// TIA Portal V20 export
FUNCTION_BLOCK "CallEquipment"   // FB44, LAD
TITLE = CallEquipment
AUTHOR : ERsystem_FA2_DH. Kim
// This block contains the logic and futher calls (e.g. sequences, control modules, diagnostics etc.) of the equipment module.
// stored: IsIECCheckEnabled true, MemoryReserve 100, Namespace Unit1.Em7, SetENOAutomatically false
   VAR_INPUT
      ZoneOperationEnable { ExternalWritable := 'False'} : "LWONIK_typeSafetyZoneManualOperation";
   END_VAR
   VAR_IN_OUT
      unitStatus : "LAF_typeUnitStatus";   // Current unit status o be used in this EM
      emFeedback : "LUC_typeEmFeedback";   // Feedback of the EM to the Unit
      unitAlarmDB : "LAF_typeAlarms";   // Summarized EM Alarms for the Unit
   END_VAR
   VAR
      instSequenceSepaClamp { ExternalAccessible := 'False'; ExternalVisible := 'False'; ExternalWritable := 'False'} : "Unit1.Em7.Sequence_1_SepaClamp";
      instSequenceSepaGripper { ExternalAccessible := 'False'; ExternalVisible := 'False'; ExternalWritable := 'False'} : "Unit1.Em7.Sequence_2_SepaGripper";
      instSequenceJellyRollWinder { ExternalAccessible := 'False'; ExternalVisible := 'False'; ExternalWritable := 'False'} : "Unit1.Em7.Sequence_3_JellyRollWinder";
      instSepaClampHomeJob1 { S7_SetPoint := 'True'} : "LAF_SelectJob";
      instSepaClampLoadJob2 { S7_SetPoint := 'True'} : "LAF_SelectJob";
      instSepaClampUnloadJob3 { S7_SetPoint := 'True'} : "LAF_SelectJob";
      instSepaClampUnloadCamJob10 { S7_SetPoint := 'True'} : "LAF_SelectJob";
      instSepaClampUnloadStopSyncJob11 { S7_SetPoint := 'True'} : "LAF_SelectJob";
      instSepaClampUnloadReturnJob12 { S7_SetPoint := 'True'} : "LAF_SelectJob";
      instSepaGripperHomeJob1 { S7_SetPoint := 'True'} : "LAF_SelectJob";
      instSepaGripperGripReadyJob2 { S7_SetPoint := 'True'} : "LAF_SelectJob";
      instSepaGripperGripSepaTailJob3 { S7_SetPoint := 'True'} : "LAF_SelectJob";
      instSepaGripperWinderMoveJob4 { S7_SetPoint := 'True'} : "LAF_SelectJob";
      instSepaGripperJellyRollUnGripJob5 { S7_SetPoint := 'True'} : "LAF_SelectJob";
      instSepaGripperJellyRollGripJob6 { S7_SetPoint := 'True'} : "LAF_SelectJob";
      instSepaGripperUnloadReadyJob7 { S7_SetPoint := 'True'} : "LAF_SelectJob";
      instSepaGripperUnloadJob8 { S7_SetPoint := 'True'} : "LAF_SelectJob";
      instSepaGripperReturnJob9 { S7_SetPoint := 'True'} : "LAF_SelectJob";
      instSepaGripperGripReadyJob11 { S7_SetPoint := 'True'} : "LAF_SelectJob";
      instSepaGripperLoadToStackTableJob12 { S7_SetPoint := 'True'} : "LAF_SelectJob";
      instSepaGripperUnLoadToJellyRollWinderJob14 { S7_SetPoint := 'True'} : "LAF_SelectJob";
      instSepaGripperLoadToJellyRollWinderJob15 { S7_SetPoint := 'True'} : "LAF_SelectJob";
      instSepaGripperUnloadToInspectionJob17 { S7_SetPoint := 'True'} : "LAF_SelectJob";
      instSepaGripperReturnJob18 { S7_SetPoint := 'True'} : "LAF_SelectJob";
      instJellyRollWinderHomeJob1 { S7_SetPoint := 'True'} : "LAF_SelectJob";
      instJellyRollWinderLoadJob2 { S7_SetPoint := 'True'} : "LAF_SelectJob";
      instJellyRollWinderWinding1Job3 { S7_SetPoint := 'True'} : "LAF_SelectJob";
      instJellyRollWinderPusherReadyJob4 { S7_SetPoint := 'True'} : "LAF_SelectJob";
      instJellyRollWinderWinding2Job5 { S7_SetPoint := 'True'} : "LAF_SelectJob";
      instJellyRollWinderUnloadJob6 { S7_SetPoint := 'True'} : "LAF_SelectJob";
      instJellyRollWinderCamWinding1stJob10 { S7_SetPoint := 'True'} : "LAF_SelectJob";
      instJellyRollWinderCamPusherReadyJob11 { S7_SetPoint := 'True'} : "LAF_SelectJob";
      instJellyRollWinderCamStartSyncJob12 { S7_SetPoint := 'True'} : "LAF_SelectJob";
      instJellyRollWinderCamWinding2ndJob13 { S7_SetPoint := 'True'} : "LAF_SelectJob";
      instJellyRollWinderCamStopSyncJob14 { S7_SetPoint := 'True'} : "LAF_SelectJob";
      instCmSepaClampDetectSensor { ExternalAccessible := 'False'; ExternalVisible := 'False'; ExternalWritable := 'False'} : "LBC_DigitalSignalCn";
      instCmSepaGripperDetectSensor { ExternalAccessible := 'False'; ExternalVisible := 'False'; ExternalWritable := 'False'} : "LBC_DigitalSignalCn";
      instCmJrWinderDetectSensor { ExternalAccessible := 'False'; ExternalVisible := 'False'; ExternalWritable := 'False'} : "LBC_DigitalSignalCn";
      instCmSepaElectrodeDetectSensor { ExternalAccessible := 'False'; ExternalVisible := 'False'; ExternalWritable := 'False'} : "LBC_DigitalSignalCn";
      instCmSepaClampSafetyPinDetectSensor { ExternalAccessible := 'False'; ExternalVisible := 'False'; ExternalWritable := 'False'} : "LBC_DigitalSignalCn";
      instCmSepaGripperSafetyPinDetectSensor { ExternalAccessible := 'False'; ExternalVisible := 'False'; ExternalWritable := 'False'} : "LBC_DigitalSignalCn";
      instCmSepaClampnCutterAxisX { ExternalAccessible := 'False'; ExternalVisible := 'False'; ExternalWritable := 'False'} : "LBC_Axis64Pos_TecPlcCn";
      instCmSepaClampnCutterAxisZ { ExternalAccessible := 'False'; ExternalVisible := 'False'; ExternalWritable := 'False'} : "LBC_Axis64Pos_TecPlcCn";
      instCmSepaGripperAxisX { ExternalAccessible := 'False'; ExternalVisible := 'False'; ExternalWritable := 'False'} : "LBC_Axis64Pos_TecPlcCn";
      instCmSepaGripperAxisZ { ExternalAccessible := 'False'; ExternalVisible := 'False'; ExternalWritable := 'False'} : "LBC_Axis64Pos_TecPlcCn";
      instCmSepaGripperAxisC { ExternalAccessible := 'False'; ExternalVisible := 'False'; ExternalWritable := 'False'} : "LBC_Axis64Pos_TecPlcCn";
      instCmJRWinderRearAxisY { ExternalAccessible := 'False'; ExternalVisible := 'False'; ExternalWritable := 'False'} : "LBC_Axis64Pos_TecPlcCn";
      instCmJRWinderFrontAxisY { ExternalAccessible := 'False'; ExternalVisible := 'False'; ExternalWritable := 'False'} : "LBC_Axis64Pos_TecPlcCn";
      instCmJRWinderAxisB { ExternalAccessible := 'False'; ExternalVisible := 'False'; ExternalWritable := 'False'} : "LBC_Axis64Pos_TecPlcCn";
      instCmJRPusherAxisZ { ExternalAccessible := 'False'; ExternalVisible := 'False'; ExternalWritable := 'False'} : "LBC_Axis64Pos_TecPlcCn";
      instInterlockSepaClampnCutterAxisX { S7_SetPoint := 'True'} : "LER_Axis64Pos_InterlockSummary";
      instInterlockSepaClampnCutterAxisZ { S7_SetPoint := 'True'} : "LER_Axis64Pos_InterlockSummary";
      instInterlockSepaGripperAxisX { S7_SetPoint := 'True'} : "LER_Axis64Pos_InterlockSummary";
      instInterlockSepaGripperAxisZ { S7_SetPoint := 'True'} : "LER_Axis64Pos_InterlockSummary";
      instInterlockSepaGripperAxisC { S7_SetPoint := 'True'} : "LER_Axis64Pos_InterlockSummary";
      instInterlockJRWinderRearAxisY { S7_SetPoint := 'True'} : "LER_Axis64Pos_InterlockSummary";
      instInterlockJRWinderFrontAxisY { S7_SetPoint := 'True'} : "LER_Axis64Pos_InterlockSummary";
      instInterlockJRWinderAxisB { S7_SetPoint := 'True'} : "LER_Axis64Pos_InterlockSummary";
      instInterlockJRPusherAxisZ { S7_SetPoint := 'True'} : "LER_Axis64Pos_InterlockSummary";
      instSepaClampAxisXCalculateCam { S7_SetPoint := 'True'} : "Unit1.Em7.SepaClampXCalculateCam";
      instSepaClampAxisZCalculateCam { S7_SetPoint := 'True'} : "Unit1.Em7.SepaClampZCalculateCam";
      instJRPusherAxisZCalculateCam { S7_SetPoint := 'True'} : "Unit1.Em7.PusherRollerZCalculateCam";
      instSepaClampAxisXMCCamIn { S7_SetPoint := 'True'} : MC_CAMIN;
      instSepaClampAxisZMCCamIn { S7_SetPoint := 'True'} : MC_CAMIN;
      instJRPusherAxisZMCCamIn { S7_SetPoint := 'True'} : MC_CAMIN;
      instCmSepaCutterUpDown { ExternalAccessible := 'False'; ExternalVisible := 'False'; ExternalWritable := 'False'} : "LBC_TwoWayActuatorCn";
      instCmSepaClampTopUpDown { ExternalAccessible := 'False'; ExternalVisible := 'False'; ExternalWritable := 'False'} : "LBC_TwoWayActuatorCn";
      instCmSepaClampBottomUpDown { ExternalAccessible := 'False'; ExternalVisible := 'False'; ExternalWritable := 'False'} : "LBC_TwoWayActuatorCn";
      instCmStackGripperOpenClose { ExternalAccessible := 'False'; ExternalVisible := 'False'; ExternalWritable := 'False'} : "LBC_TwoWayActuatorCn";
      instCmStackGripperFwdBwd { ExternalAccessible := 'False'; ExternalVisible := 'False'; ExternalWritable := 'False'} : "LBC_TwoWayActuatorCn";
      instCmJRWinderClampTopRearUpDown { ExternalAccessible := 'False'; ExternalVisible := 'False'; ExternalWritable := 'False'} : "LBC_TwoWayActuatorCn";
      instCmJRWinderClampBtmRearUpDown { ExternalAccessible := 'False'; ExternalVisible := 'False'; ExternalWritable := 'False'} : "LBC_TwoWayActuatorCn";
      instCmJRWinderClampTopFrontUpDown { ExternalAccessible := 'False'; ExternalVisible := 'False'; ExternalWritable := 'False'} : "LBC_TwoWayActuatorCn";
      instCmJRWinderClampBtmFrontUpDown { ExternalAccessible := 'False'; ExternalVisible := 'False'; ExternalWritable := 'False'} : "LBC_TwoWayActuatorCn";
      instCmPusherRollerFwdBwd { ExternalAccessible := 'False'; ExternalVisible := 'False'; ExternalWritable := 'False'} : "LBC_TwoWayActuatorCn";
      instManageAlarms { ExternalAccessible := 'False'; ExternalVisible := 'False'; ExternalWritable := 'False'} : "LAF_ManageAlarms";
      instEventsPFE { ExternalAccessible := 'False'; ExternalVisible := 'False'; ExternalWritable := 'False'} : "Unit1.Em7.EventsPFE";
      instLER_BrakeTestSepaClampNCutterAxisZ : "LER_BrakeTest";
      instLER_BrakeTestSepaGripperAxisZ { S7_SetPoint := 'True'} : "LER_BrakeTest";
      instLER_BrakeTestJRPusherAxisZ { S7_SetPoint := 'True'} : "LER_BrakeTest";
      statUnitStatus { ExternalAccessible := 'False'; ExternalVisible := 'False'; ExternalWritable := 'False'} : "LAF_typeUnitStatus";   // Unit Status used in this EM
      statSlmStatus : Struct
         running { ExternalWritable := 'False'} : Bool;
         powerOff { ExternalWritable := 'False'} : Bool;
      END_STRUCT;
      statAllBrakeTest { ExternalWritable := 'False'} : "LER_typeBrakeTestUnitCommands";
      statTonTime { ExternalAccessible := 'False'; ExternalVisible := 'False'; ExternalWritable := 'False'} : Array[0..1999] of TON_TIME;
      statTofTime { ExternalAccessible := 'False'; ExternalVisible := 'False'; ExternalWritable := 'False'} : Array[0..99] of TOF_TIME;
      statPulse { ExternalAccessible := 'False'; ExternalVisible := 'False'; ExternalWritable := 'False'} : Struct
         miscellaneous : Array[0..99] of Bool;
         workingDone : Struct
            sepaClamp : Array[0..99] of Bool;
            sepaGripper : Array[0..99] of Bool;
            winder : Array[0..99] of Bool;
         END_STRUCT;
         axisEnable : Array[0..99] of Bool;
         brakeTest : Array[0..99] of Bool;
      END_STRUCT;
      statEnableManualCmds { ExternalAccessible := 'False'; ExternalVisible := 'False'; ExternalWritable := 'False'} : Bool;
      scan_on : Bool;
      "*** Interlock Axis ***" { ExternalAccessible := 'False'; ExternalVisible := 'False'; ExternalWritable := 'False'} : Bool;
      instSepaClampnCutterAxisX_CW { S7_SetPoint := 'True'} : "Jog.LER_Axis";
      instSepaClampnCutterAxisX_CCW { S7_SetPoint := 'True'} : "Jog.LER_Axis";
      instSepaClampnCutterAxisX_Home { S7_SetPoint := 'True'} : "Homing.LER_Axis";
      instSepaClampnCutterAxisX_Position { S7_SetPoint := 'True'} : Array[0..6] of "Position.LER_Axis";
      instSepaClampnCutterAxisZ_CW { S7_SetPoint := 'True'} : "Jog.LER_Axis";
      instSepaClampnCutterAxisZ_CCW { S7_SetPoint := 'True'} : "Jog.LER_Axis";
      instSepaClampnCutterAxisZ_Home { S7_SetPoint := 'True'} : "Homing.LER_Axis";
      instSepaClampnCutterAxisZ_Position { S7_SetPoint := 'True'} : Array[0..6] of "Position.LER_Axis";
      instSepaGripperAxisX_CW { S7_SetPoint := 'True'} : "Jog.LER_Axis";
      instSepaGripperAxisX_CCW { S7_SetPoint := 'True'} : "Jog.LER_Axis";
      instSepaGripperAxisX_Home { S7_SetPoint := 'True'} : "Homing.LER_Axis";
      instSepaGripperAxisX_Position { S7_SetPoint := 'True'} : Array[0..15] of "Position.LER_Axis";
      instSepaGripperAxisZ_CW { S7_SetPoint := 'True'} : "Jog.LER_Axis";
      instSepaGripperAxisZ_CCW { S7_SetPoint := 'True'} : "Jog.LER_Axis";
      instSepaGripperAxisZ_Home { S7_SetPoint := 'True'} : "Homing.LER_Axis";
      instSepaGripperAxisZ_Position { S7_SetPoint := 'True'} : Array[0..6] of "Position.LER_Axis";
      instSepaGripperAxisC_CW { S7_SetPoint := 'True'} : "Jog.LER_Axis";
      instSepaGripperAxisC_CCW { S7_SetPoint := 'True'} : "Jog.LER_Axis";
      instSepaGripperAxisC_Home { S7_SetPoint := 'True'} : "Homing.LER_Axis";
      instSepaGripperAxisC_Position { S7_SetPoint := 'True'} : Array[0..6] of "Position.LER_Axis";
      instJRWinderRearAxisY_CW { S7_SetPoint := 'True'} : "Jog.LER_Axis";
      instJRWinderRearAxisY_CCW { S7_SetPoint := 'True'} : "Jog.LER_Axis";
      instJRWinderRearAxisY_Home { S7_SetPoint := 'True'} : "Homing.LER_Axis";
      instJRWinderRearAxisY_Position { S7_SetPoint := 'True'} : Array[0..6] of "Position.LER_Axis";
      instJRWinderFrontAxisY_CW { S7_SetPoint := 'True'} : "Jog.LER_Axis";
      instJRWinderFrontAxisY_CCW { S7_SetPoint := 'True'} : "Jog.LER_Axis";
      instJRWinderFrontAxisY_Home { S7_SetPoint := 'True'} : "Homing.LER_Axis";
      instJRWinderFrontAxisY_Position { S7_SetPoint := 'True'} : Array[0..6] of "Position.LER_Axis";
      instJRWinderAxisB_CW { S7_SetPoint := 'True'} : "Jog.LER_Axis";
      instJRWinderAxisB_CCW { S7_SetPoint := 'True'} : "Jog.LER_Axis";
      instJRWinderAxisB_Home { S7_SetPoint := 'True'} : "Homing.LER_Axis";
      instJRWinderAxisB_Position { S7_SetPoint := 'True'} : Array[0..8] of "Position.LER_Axis";
      instJRPusherAxisZ_CW { S7_SetPoint := 'True'} : "Jog.LER_Axis";
      instJRPusherAxisZ_CCW { S7_SetPoint := 'True'} : "Jog.LER_Axis";
      instJRPusherAxisZ_Home { S7_SetPoint := 'True'} : "Homing.LER_Axis";
      instJRPusherAxisZ_Position { S7_SetPoint := 'True'} : Array[0..6] of "Position.LER_Axis";
      "*** Interlock Actuator ******" { ExternalAccessible := 'False'; ExternalVisible := 'False'; ExternalWritable := 'False'} : Bool;
      instCmSepaCutterUpDownInterlock : Array[0..1] of "Cylinder.LER_Actuator";
      instCmSepaClampTopUpDownInterlock { S7_SetPoint := 'True'} : Array[0..1] of "Cylinder.LER_Actuator";
      instCmSepaClampBottomUpDownInterlock { S7_SetPoint := 'True'} : Array[0..1] of "Cylinder.LER_Actuator";
      instCmStackGripperOpenCloseInterlock { S7_SetPoint := 'True'} : Array[0..1] of "Cylinder.LER_Actuator";
      instCmStackGripperFwdBwdInterlock { S7_SetPoint := 'True'} : Array[0..1] of "Cylinder.LER_Actuator";
      instCmJRWinderClampTopRearUpDownInterlock { S7_SetPoint := 'True'} : Array[0..1] of "Cylinder.LER_Actuator";
      instCmJRWinderClampBtmRearUpDownInterlock { S7_SetPoint := 'True'} : Array[0..1] of "Cylinder.LER_Actuator";
      instCmJRWinderClampTopFrontUpDownInterlock { S7_SetPoint := 'True'} : Array[0..1] of "Cylinder.LER_Actuator";
      instCmJRWinderClampBtmFrontUpDownInterlock { S7_SetPoint := 'True'} : Array[0..1] of "Cylinder.LER_Actuator";
      instCmPusherRollerFwdBwdInterlock { S7_SetPoint := 'True'} : Array[0..1] of "Cylinder.LER_Actuator";
      Tracking_07 { S7_SetPoint := 'True'} : "Unit1.Em7.PartData";
      AXIS34 : "LER_CM_Name";
      AXIS39 : "LER_CM_Name";
      Cylinder38 : "LER_CM_Name";
      Cylinder43 : "LER_CM_Name";
      citi_Ptrig : Array[0..20] of Bool;
      citiTon : Array[0..20] of TON_TIME;
      citi : Time;
      citiTest : Array[0..20] of Bool;
   END_VAR
   VAR_TEMP
      tempScInProduction : Bool;   // Mode Production and StateComplete
      tempScNoProduction : Bool;   // Mode Manual and StateComplete
   END_VAR
   VAR CONSTANT
      delayTime : Time := T#3s;
      TRUE : Bool := TRUE;
      FALSE : Bool := FALSE;
      NO_JOB : DInt;   // No job
      MIN_POSITION_NUMBER : SInt;
      INIT_POSITION_NUMBER : SInt := -1;
   END_VAR
   // // statPulse.brakeTest[0] : Unit Mode Production Rising Edge
   // // statPulse.brakeTest[1] : Unit Mode Production Rising Edge Old
   // // statPulse.brakeTest[10] : Sepa Clamp Cutter Z Axis Error Pulse
   // // statPulse.brakeTest[11] : Sepa Gripper Z Axis Error Pulse
   // // statPulse.brakeTest[12] : JR Pusher Z Axis Error Pulse
   VAR_TEMP   // added for the SCL form of the ladder/FBD networks
      _w1 : Bool;
      _w2 : Bool;
      _w3 : Bool;
      _w4 : Bool;
      _w5 : Bool;
      _w6 : Bool;
      _w7 : Bool;
      _w8 : Bool;
      _w9 : Bool;
      _w10 : Bool;
      _w11 : Bool;
   END_VAR
BEGIN

REGION Network 1: BLOCK INFO HEADER
   // (company) / (C) Copyright (year)
   // ---------------------------------------------------------------------------------
   // Title:                             (Title of this block)
   // Comment/Function: (that is implemented in the block)
   // Library/Family:           (that the source is dedicated to)
   // Author:                        (department / person in charge / contact)
   // Target System:          (test system with FW version)
   // Engineering:              TIA Portal (SW version)
   // Restrictions:               (OB types, etc.)
   // Requirements:           (hardware, technological package, etc.)
   // ---------------------------------------------------------------------------------
   // Change log table:
   // Version          | Date             | Signature      | Expert in charge  | Changes applied ------------------------|----------------------|-------------------------|--------------------------------|-----------------------
   // 001.000.000 | yyyy-mm-dd | 0x00000000 | (name of expert) | First released version
END_REGION

REGION Network 2: DESCRIPTION
   // This is a template block provided by the Automation Framework. It can be used to create an own project.
   // The Block Info Header is prepared to put in your own data.
   // Description of the block could be added here and the docu created by Code2Docu.
END_REGION

REGION Network 3: TRUE: Disable the monitoring of the Home position feedback. FALSE: Home position is reached after `monitoringReachingFeedback` time expires.
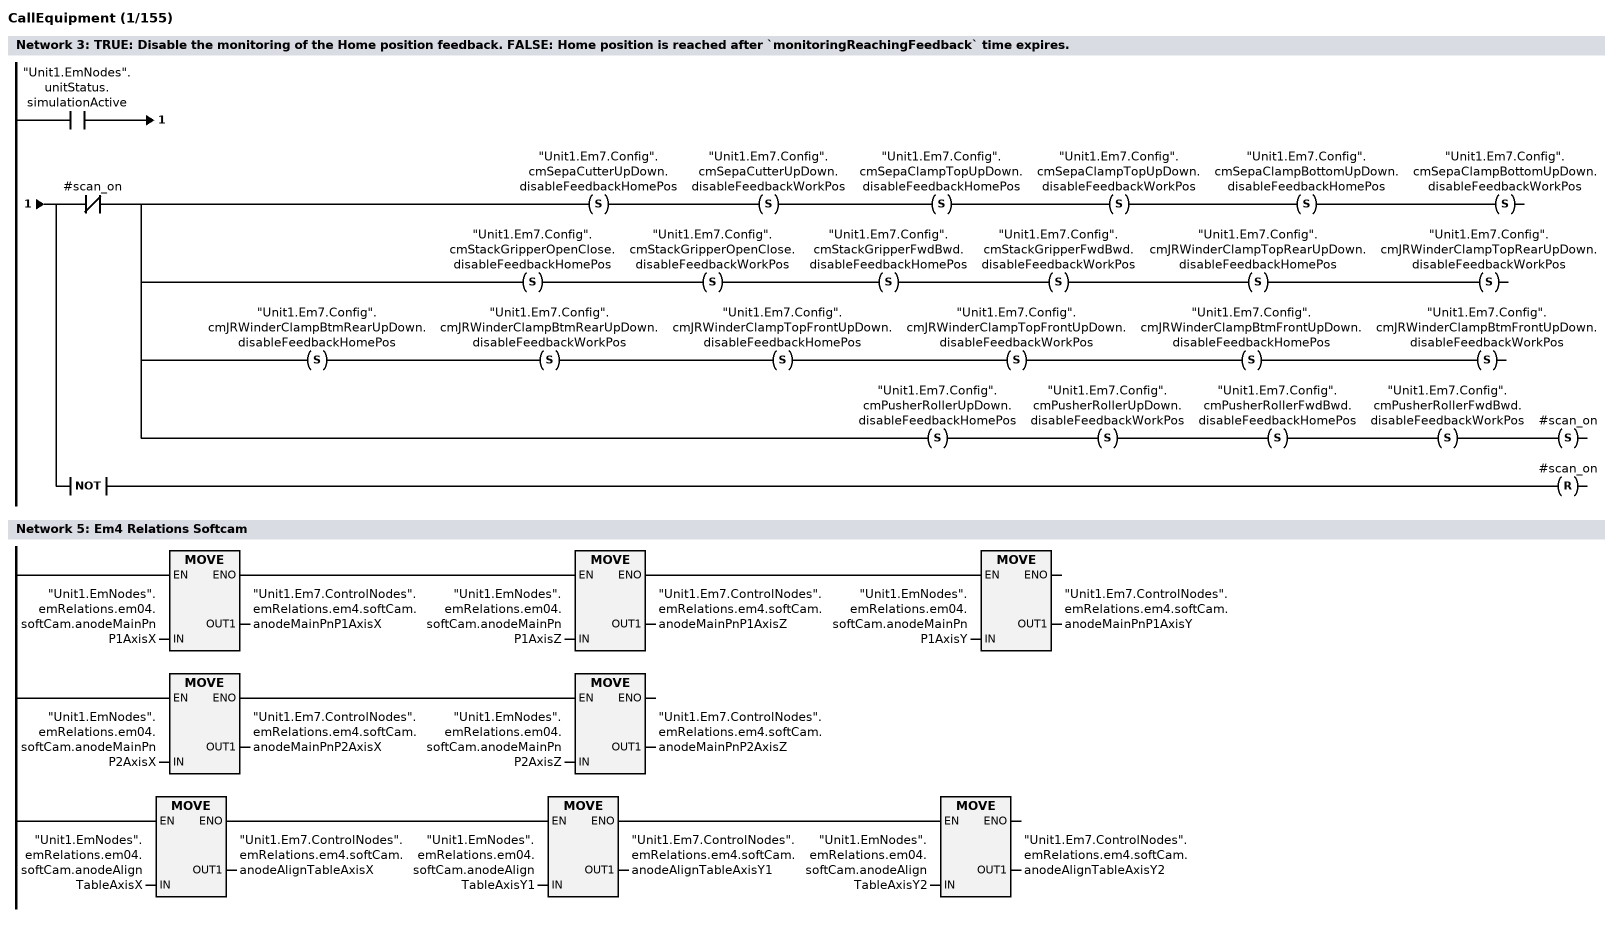
   RUNG wire#powerrail
      Contact( "Unit1.EmNodes".unitStatus.simulationActive )
      wire#w1
      I_Contact( #scan_on )
      wire#w2
      S_Coil( "Unit1.Em7.Config".cmSepaCutterUpDown.disableFeedbackHomePos )
      S_Coil( "Unit1.Em7.Config".cmSepaCutterUpDown.disableFeedbackWorkPos )
      S_Coil( "Unit1.Em7.Config".cmSepaClampTopUpDown.disableFeedbackHomePos )
      S_Coil( "Unit1.Em7.Config".cmSepaClampTopUpDown.disableFeedbackWorkPos )
      S_Coil( "Unit1.Em7.Config".cmSepaClampBottomUpDown.disableFeedbackHomePos )
      S_Coil( "Unit1.Em7.Config".cmSepaClampBottomUpDown.disableFeedbackWorkPos )
   END_RUNG
   RUNG wire#w2
      S_Coil( "Unit1.Em7.Config".cmStackGripperOpenClose.disableFeedbackHomePos )
      S_Coil( "Unit1.Em7.Config".cmStackGripperOpenClose.disableFeedbackWorkPos )
      S_Coil( "Unit1.Em7.Config".cmStackGripperFwdBwd.disableFeedbackHomePos )
      S_Coil( "Unit1.Em7.Config".cmStackGripperFwdBwd.disableFeedbackWorkPos )
      S_Coil( "Unit1.Em7.Config".cmJRWinderClampTopRearUpDown.disableFeedbackHomePos )
      S_Coil( "Unit1.Em7.Config".cmJRWinderClampTopRearUpDown.disableFeedbackWorkPos )
   END_RUNG
   RUNG wire#w2
      S_Coil( "Unit1.Em7.Config".cmJRWinderClampBtmRearUpDown.disableFeedbackHomePos )
      S_Coil( "Unit1.Em7.Config".cmJRWinderClampBtmRearUpDown.disableFeedbackWorkPos )
      S_Coil( "Unit1.Em7.Config".cmJRWinderClampTopFrontUpDown.disableFeedbackHomePos )
      S_Coil( "Unit1.Em7.Config".cmJRWinderClampTopFrontUpDown.disableFeedbackWorkPos )
      S_Coil( "Unit1.Em7.Config".cmJRWinderClampBtmFrontUpDown.disableFeedbackHomePos )
      S_Coil( "Unit1.Em7.Config".cmJRWinderClampBtmFrontUpDown.disableFeedbackWorkPos )
   END_RUNG
   RUNG wire#w2
      S_Coil( "Unit1.Em7.Config".cmPusherRollerUpDown.disableFeedbackHomePos )
      S_Coil( "Unit1.Em7.Config".cmPusherRollerUpDown.disableFeedbackWorkPos )
      S_Coil( "Unit1.Em7.Config".cmPusherRollerFwdBwd.disableFeedbackHomePos )
      S_Coil( "Unit1.Em7.Config".cmPusherRollerFwdBwd.disableFeedbackWorkPos )
      S_Coil( #scan_on )
   END_RUNG
   RUNG wire#w1
      Not()
      R_Coil( #scan_on )
   END_RUNG
   // the same network as SCL:
   IF "Unit1.EmNodes".unitStatus.simulationActive AND NOT #scan_on THEN
       "Unit1.Em7.Config".cmSepaCutterUpDown.disableFeedbackHomePos := TRUE;
       "Unit1.Em7.Config".cmSepaCutterUpDown.disableFeedbackWorkPos := TRUE;
       "Unit1.Em7.Config".cmSepaClampTopUpDown.disableFeedbackHomePos := TRUE;
       "Unit1.Em7.Config".cmSepaClampTopUpDown.disableFeedbackWorkPos := TRUE;
       "Unit1.Em7.Config".cmSepaClampBottomUpDown.disableFeedbackHomePos := TRUE;
       "Unit1.Em7.Config".cmSepaClampBottomUpDown.disableFeedbackWorkPos := TRUE;
       "Unit1.Em7.Config".cmStackGripperOpenClose.disableFeedbackHomePos := TRUE;
       "Unit1.Em7.Config".cmStackGripperOpenClose.disableFeedbackWorkPos := TRUE;
       "Unit1.Em7.Config".cmStackGripperFwdBwd.disableFeedbackHomePos := TRUE;
       "Unit1.Em7.Config".cmStackGripperFwdBwd.disableFeedbackWorkPos := TRUE;
       "Unit1.Em7.Config".cmJRWinderClampTopRearUpDown.disableFeedbackHomePos := TRUE;
       "Unit1.Em7.Config".cmJRWinderClampTopRearUpDown.disableFeedbackWorkPos := TRUE;
       "Unit1.Em7.Config".cmJRWinderClampBtmRearUpDown.disableFeedbackHomePos := TRUE;
       "Unit1.Em7.Config".cmJRWinderClampBtmRearUpDown.disableFeedbackWorkPos := TRUE;
       "Unit1.Em7.Config".cmJRWinderClampTopFrontUpDown.disableFeedbackHomePos := TRUE;
       "Unit1.Em7.Config".cmJRWinderClampTopFrontUpDown.disableFeedbackWorkPos := TRUE;
       "Unit1.Em7.Config".cmJRWinderClampBtmFrontUpDown.disableFeedbackHomePos := TRUE;
       "Unit1.Em7.Config".cmJRWinderClampBtmFrontUpDown.disableFeedbackWorkPos := TRUE;
       "Unit1.Em7.Config".cmPusherRollerUpDown.disableFeedbackHomePos := TRUE;
       "Unit1.Em7.Config".cmPusherRollerUpDown.disableFeedbackWorkPos := TRUE;
       "Unit1.Em7.Config".cmPusherRollerFwdBwd.disableFeedbackHomePos := TRUE;
       "Unit1.Em7.Config".cmPusherRollerFwdBwd.disableFeedbackWorkPos := TRUE;
       #scan_on := TRUE;
   END_IF;
   IF NOT "Unit1.EmNodes".unitStatus.simulationActive THEN #scan_on := FALSE; END_IF;
END_REGION

REGION Network 4: ******************** Unit Input ********************
END_REGION

REGION Network 5: Em4 Relations Softcam
   RUNG wire#powerrail
      Move(in := "Unit1.EmNodes".emRelations.em04.softCam.anodeMainPnP1AxisX, out1 => "Unit1.Em7.ControlNodes".emRelations.em4.softCam.anodeMainPnP1AxisX)
      Move(in := "Unit1.EmNodes".emRelations.em04.softCam.anodeMainPnP1AxisZ, out1 => "Unit1.Em7.ControlNodes".emRelations.em4.softCam.anodeMainPnP1AxisZ)
      Move(in := "Unit1.EmNodes".emRelations.em04.softCam.anodeMainPnP1AxisY, out1 => "Unit1.Em7.ControlNodes".emRelations.em4.softCam.anodeMainPnP1AxisY)
   END_RUNG
   RUNG wire#powerrail
      Move(in := "Unit1.EmNodes".emRelations.em04.softCam.anodeMainPnP2AxisX, out1 => "Unit1.Em7.ControlNodes".emRelations.em4.softCam.anodeMainPnP2AxisX)
      Move(in := "Unit1.EmNodes".emRelations.em04.softCam.anodeMainPnP2AxisZ, out1 => "Unit1.Em7.ControlNodes".emRelations.em4.softCam.anodeMainPnP2AxisZ)
   END_RUNG
   RUNG wire#powerrail
      Move(in := "Unit1.EmNodes".emRelations.em04.softCam.anodeAlignTableAxisX, out1 => "Unit1.Em7.ControlNodes".emRelations.em4.softCam.anodeAlignTableAxisX)
      Move(in := "Unit1.EmNodes".emRelations.em04.softCam.anodeAlignTableAxisY1, out1 => "Unit1.Em7.ControlNodes".emRelations.em4.softCam.anodeAlignTableAxisY1)
      Move(in := "Unit1.EmNodes".emRelations.em04.softCam.anodeAlignTableAxisY2, out1 => "Unit1.Em7.ControlNodes".emRelations.em4.softCam.anodeAlignTableAxisY2)
   END_RUNG
   // the same network as SCL:
   "Unit1.Em7.ControlNodes".emRelations.em4.softCam.anodeMainPnP1AxisX := "Unit1.EmNodes".emRelations.em04.softCam.anodeMainPnP1AxisX;
   "Unit1.Em7.ControlNodes".emRelations.em4.softCam.anodeMainPnP1AxisZ := "Unit1.EmNodes".emRelations.em04.softCam.anodeMainPnP1AxisZ;
   "Unit1.Em7.ControlNodes".emRelations.em4.softCam.anodeMainPnP1AxisY := "Unit1.EmNodes".emRelations.em04.softCam.anodeMainPnP1AxisY;
   "Unit1.Em7.ControlNodes".emRelations.em4.softCam.anodeMainPnP2AxisX := "Unit1.EmNodes".emRelations.em04.softCam.anodeMainPnP2AxisX;
   "Unit1.Em7.ControlNodes".emRelations.em4.softCam.anodeMainPnP2AxisZ := "Unit1.EmNodes".emRelations.em04.softCam.anodeMainPnP2AxisZ;
   "Unit1.Em7.ControlNodes".emRelations.em4.softCam.anodeAlignTableAxisX := "Unit1.EmNodes".emRelations.em04.softCam.anodeAlignTableAxisX;
   "Unit1.Em7.ControlNodes".emRelations.em4.softCam.anodeAlignTableAxisY1 := "Unit1.EmNodes".emRelations.em04.softCam.anodeAlignTableAxisY1;
   "Unit1.Em7.ControlNodes".emRelations.em4.softCam.anodeAlignTableAxisY2 := "Unit1.EmNodes".emRelations.em04.softCam.anodeAlignTableAxisY2;
END_REGION

REGION Network 6: Em6 Relations Softcam
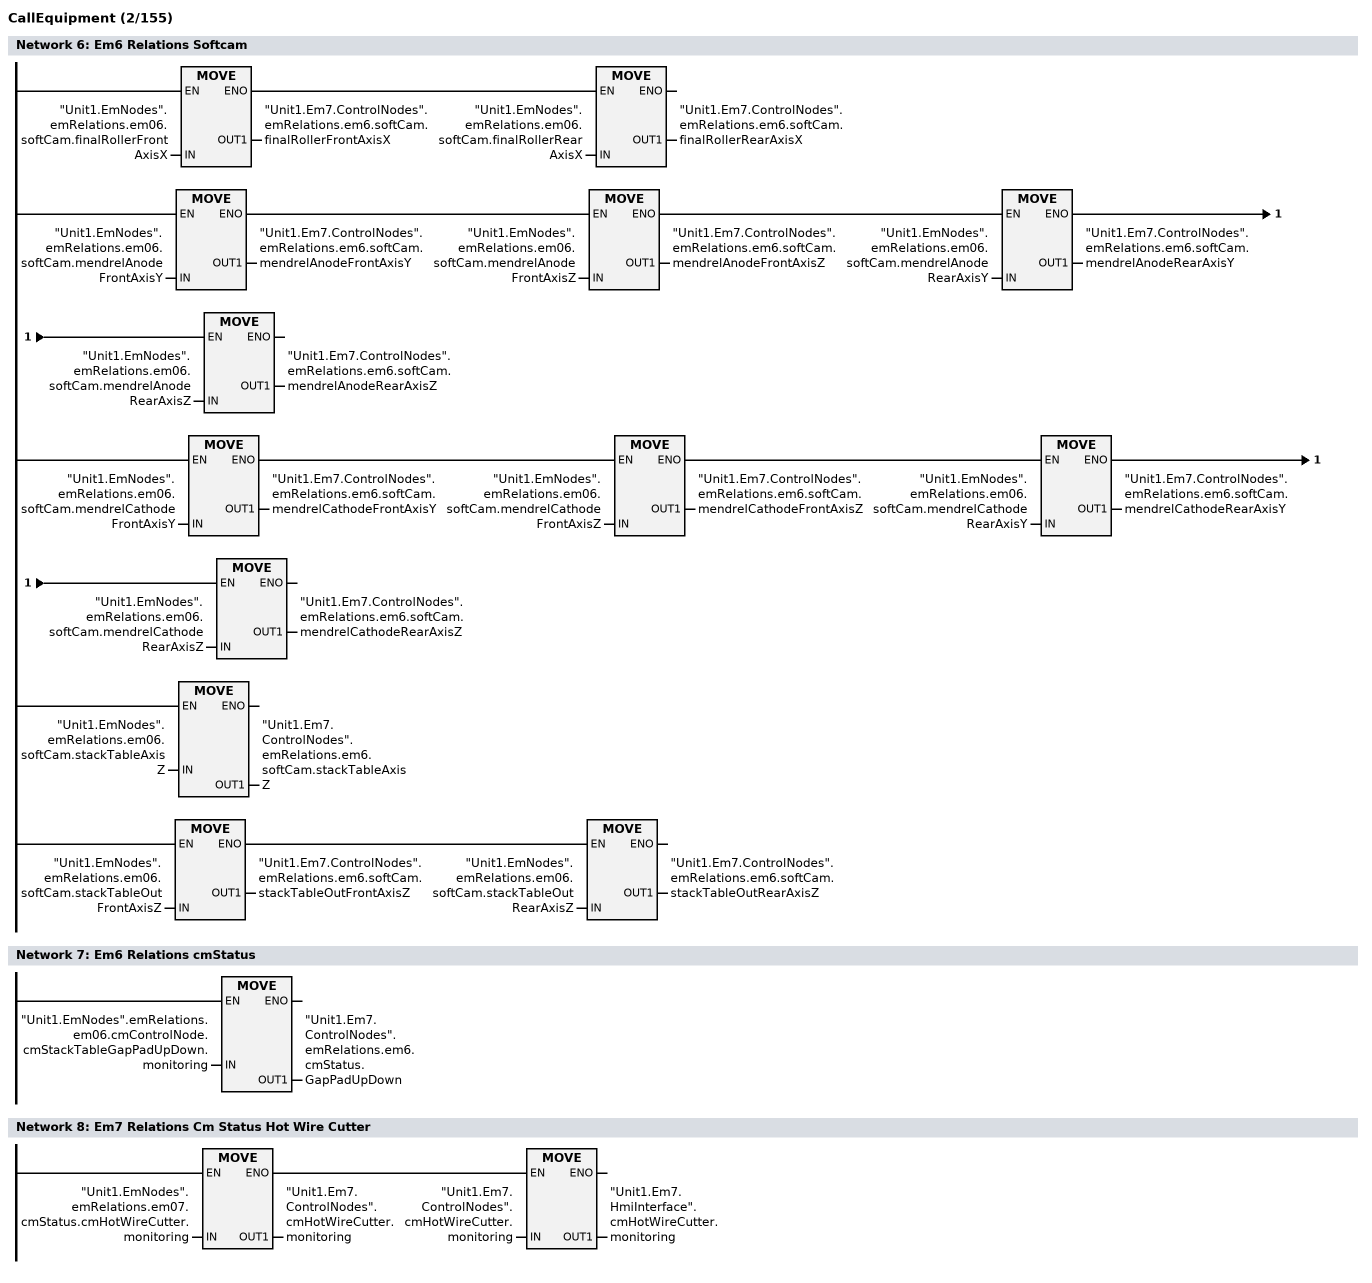
   RUNG wire#powerrail
      Move(in := "Unit1.EmNodes".emRelations.em06.softCam.finalRollerFrontAxisX, out1 => "Unit1.Em7.ControlNodes".emRelations.em6.softCam.finalRollerFrontAxisX)
      Move(in := "Unit1.EmNodes".emRelations.em06.softCam.finalRollerRearAxisX, out1 => "Unit1.Em7.ControlNodes".emRelations.em6.softCam.finalRollerRearAxisX)
   END_RUNG
   RUNG wire#powerrail
      Move(in := "Unit1.EmNodes".emRelations.em06.softCam.mendrelAnodeFrontAxisY, out1 => "Unit1.Em7.ControlNodes".emRelations.em6.softCam.mendrelAnodeFrontAxisY)
      Move(in := "Unit1.EmNodes".emRelations.em06.softCam.mendrelAnodeFrontAxisZ, out1 => "Unit1.Em7.ControlNodes".emRelations.em6.softCam.mendrelAnodeFrontAxisZ)
      Move(in := "Unit1.EmNodes".emRelations.em06.softCam.mendrelAnodeRearAxisY, out1 => "Unit1.Em7.ControlNodes".emRelations.em6.softCam.mendrelAnodeRearAxisY)
      Move(in := "Unit1.EmNodes".emRelations.em06.softCam.mendrelAnodeRearAxisZ, out1 => "Unit1.Em7.ControlNodes".emRelations.em6.softCam.mendrelAnodeRearAxisZ)
   END_RUNG
   RUNG wire#powerrail
      Move(in := "Unit1.EmNodes".emRelations.em06.softCam.mendrelCathodeFrontAxisY, out1 => "Unit1.Em7.ControlNodes".emRelations.em6.softCam.mendrelCathodeFrontAxisY)
      Move(in := "Unit1.EmNodes".emRelations.em06.softCam.mendrelCathodeFrontAxisZ, out1 => "Unit1.Em7.ControlNodes".emRelations.em6.softCam.mendrelCathodeFrontAxisZ)
      Move(in := "Unit1.EmNodes".emRelations.em06.softCam.mendrelCathodeRearAxisY, out1 => "Unit1.Em7.ControlNodes".emRelations.em6.softCam.mendrelCathodeRearAxisY)
      Move(in := "Unit1.EmNodes".emRelations.em06.softCam.mendrelCathodeRearAxisZ, out1 => "Unit1.Em7.ControlNodes".emRelations.em6.softCam.mendrelCathodeRearAxisZ)
   END_RUNG
   RUNG wire#powerrail
      Move(in := "Unit1.EmNodes".emRelations.em06.softCam.stackTableAxisZ, out1 => "Unit1.Em7.ControlNodes".emRelations.em6.softCam.stackTableAxisZ)
   END_RUNG
   RUNG wire#powerrail
      Move(in := "Unit1.EmNodes".emRelations.em06.softCam.stackTableOutFrontAxisZ, out1 => "Unit1.Em7.ControlNodes".emRelations.em6.softCam.stackTableOutFrontAxisZ)
      Move(in := "Unit1.EmNodes".emRelations.em06.softCam.stackTableOutRearAxisZ, out1 => "Unit1.Em7.ControlNodes".emRelations.em6.softCam.stackTableOutRearAxisZ)
   END_RUNG
   // the same network as SCL:
   "Unit1.Em7.ControlNodes".emRelations.em6.softCam.finalRollerFrontAxisX := "Unit1.EmNodes".emRelations.em06.softCam.finalRollerFrontAxisX;
   "Unit1.Em7.ControlNodes".emRelations.em6.softCam.finalRollerRearAxisX := "Unit1.EmNodes".emRelations.em06.softCam.finalRollerRearAxisX;
   "Unit1.Em7.ControlNodes".emRelations.em6.softCam.mendrelAnodeFrontAxisY := "Unit1.EmNodes".emRelations.em06.softCam.mendrelAnodeFrontAxisY;
   "Unit1.Em7.ControlNodes".emRelations.em6.softCam.mendrelAnodeFrontAxisZ := "Unit1.EmNodes".emRelations.em06.softCam.mendrelAnodeFrontAxisZ;
   "Unit1.Em7.ControlNodes".emRelations.em6.softCam.mendrelAnodeRearAxisY := "Unit1.EmNodes".emRelations.em06.softCam.mendrelAnodeRearAxisY;
   "Unit1.Em7.ControlNodes".emRelations.em6.softCam.mendrelAnodeRearAxisZ := "Unit1.EmNodes".emRelations.em06.softCam.mendrelAnodeRearAxisZ;
   "Unit1.Em7.ControlNodes".emRelations.em6.softCam.mendrelCathodeFrontAxisY := "Unit1.EmNodes".emRelations.em06.softCam.mendrelCathodeFrontAxisY;
   "Unit1.Em7.ControlNodes".emRelations.em6.softCam.mendrelCathodeFrontAxisZ := "Unit1.EmNodes".emRelations.em06.softCam.mendrelCathodeFrontAxisZ;
   "Unit1.Em7.ControlNodes".emRelations.em6.softCam.mendrelCathodeRearAxisY := "Unit1.EmNodes".emRelations.em06.softCam.mendrelCathodeRearAxisY;
   "Unit1.Em7.ControlNodes".emRelations.em6.softCam.mendrelCathodeRearAxisZ := "Unit1.EmNodes".emRelations.em06.softCam.mendrelCathodeRearAxisZ;
   "Unit1.Em7.ControlNodes".emRelations.em6.softCam.stackTableAxisZ := "Unit1.EmNodes".emRelations.em06.softCam.stackTableAxisZ;
   "Unit1.Em7.ControlNodes".emRelations.em6.softCam.stackTableOutFrontAxisZ := "Unit1.EmNodes".emRelations.em06.softCam.stackTableOutFrontAxisZ;
   "Unit1.Em7.ControlNodes".emRelations.em6.softCam.stackTableOutRearAxisZ := "Unit1.EmNodes".emRelations.em06.softCam.stackTableOutRearAxisZ;
END_REGION

REGION Network 7: Em6 Relations cmStatus
   RUNG wire#powerrail
      Move(in := "Unit1.EmNodes".emRelations.em06.cmControlNode.cmStackTableGapPadUpDown.monitoring, out1 => "Unit1.Em7.ControlNodes".emRelations.em6.cmStatus.GapPadUpDown)
   END_RUNG
   // the same network as SCL:
   "Unit1.Em7.ControlNodes".emRelations.em6.cmStatus.GapPadUpDown := "Unit1.EmNodes".emRelations.em06.cmControlNode.cmStackTableGapPadUpDown.monitoring;
END_REGION

REGION Network 8: Em7 Relations Cm Status Hot Wire Cutter
   RUNG wire#powerrail
      Move(in := "Unit1.EmNodes".emRelations.em07.cmStatus.cmHotWireCutter.monitoring, out1 => "Unit1.Em7.ControlNodes".cmHotWireCutter.monitoring)
      Move(in := "Unit1.Em7.ControlNodes".cmHotWireCutter.monitoring, out1 => "Unit1.Em7.HmiInterface".cmHotWireCutter.monitoring)
   END_RUNG
   // the same network as SCL:
   "Unit1.Em7.ControlNodes".cmHotWireCutter.monitoring := "Unit1.EmNodes".emRelations.em07.cmStatus.cmHotWireCutter.monitoring;
   "Unit1.Em7.HmiInterface".cmHotWireCutter.monitoring := "Unit1.Em7.ControlNodes".cmHotWireCutter.monitoring;
END_REGION

REGION Network 9: Em Nodes BA060 Communication
END_REGION

REGION Network 10: Em Nodes Power Status
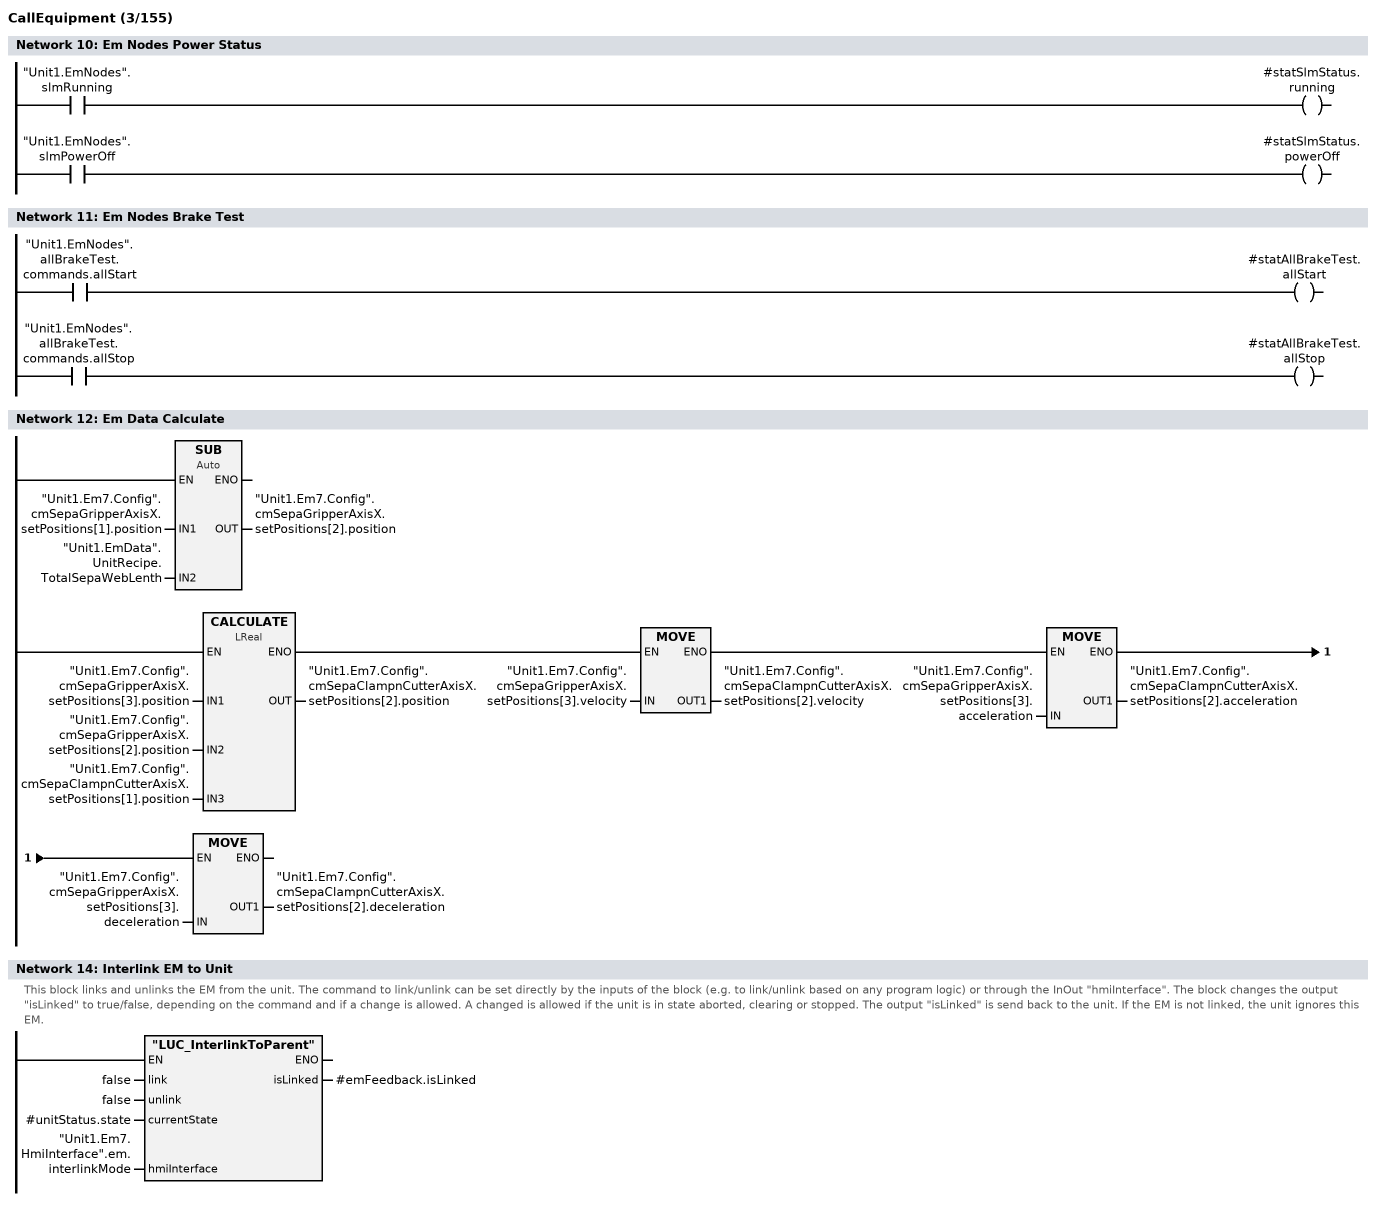
   RUNG wire#powerrail
      Contact( "Unit1.EmNodes".slmRunning )
      Coil( #statSlmStatus.running )
   END_RUNG
   RUNG wire#powerrail
      Contact( "Unit1.EmNodes".slmPowerOff )
      Coil( #statSlmStatus.powerOff )
   END_RUNG
   // the same network as SCL:
   #statSlmStatus.running := "Unit1.EmNodes".slmRunning;
   #statSlmStatus.powerOff := "Unit1.EmNodes".slmPowerOff;
END_REGION

REGION Network 11: Em Nodes Brake Test
   RUNG wire#powerrail
      Contact( "Unit1.EmNodes".allBrakeTest.commands.allStart )
      Coil( #statAllBrakeTest.allStart )
   END_RUNG
   RUNG wire#powerrail
      Contact( "Unit1.EmNodes".allBrakeTest.commands.allStop )
      Coil( #statAllBrakeTest.allStop )
   END_RUNG
   // the same network as SCL:
   #statAllBrakeTest.allStart := "Unit1.EmNodes".allBrakeTest.commands.allStart;
   #statAllBrakeTest.allStop := "Unit1.EmNodes".allBrakeTest.commands.allStop;
END_REGION

REGION Network 12: Em Data Calculate
   RUNG wire#powerrail
      Sub(in1 := "Unit1.Em7.Config".cmSepaGripperAxisX.setPositions[1].position, in2 := "Unit1.EmData".UnitRecipe.TotalSepaWebLenth, out => "Unit1.Em7.Config".cmSepaGripperAxisX.setPositions[2].position)
   END_RUNG
   RUNG wire#powerrail
      { S7_Templates := "SrcType := LReal"; S7_Expression := "IN2-IN1+IN3" } Calculate(in1 := "Unit1.Em7.Config".cmSepaGripperAxisX.setPositions[3].position, in2 := "Unit1.Em7.Config".cmSepaGripperAxisX.setPositions[2].position, in3 := "Unit1.Em7.Config".cmSepaClampnCutterAxisX.setPositions[1].position, out => "Unit1.Em7.Config".cmSepaClampnCutterAxisX.setPositions[2].position)
      Move(in := "Unit1.Em7.Config".cmSepaGripperAxisX.setPositions[3].velocity, out1 => "Unit1.Em7.Config".cmSepaClampnCutterAxisX.setPositions[2].velocity)
      Move(in := "Unit1.Em7.Config".cmSepaGripperAxisX.setPositions[3].acceleration, out1 => "Unit1.Em7.Config".cmSepaClampnCutterAxisX.setPositions[2].acceleration)
      Move(in := "Unit1.Em7.Config".cmSepaGripperAxisX.setPositions[3].deceleration, out1 => "Unit1.Em7.Config".cmSepaClampnCutterAxisX.setPositions[2].deceleration)
   END_RUNG
   // the same network as SCL:
   "Unit1.Em7.Config".cmSepaGripperAxisX.setPositions[2].position := "Unit1.Em7.Config".cmSepaGripperAxisX.setPositions[1].position - "Unit1.EmData".UnitRecipe.TotalSepaWebLenth;
   "Unit1.Em7.Config".cmSepaClampnCutterAxisX.setPositions[2].position := "Unit1.Em7.Config".cmSepaGripperAxisX.setPositions[2].position-"Unit1.Em7.Config".cmSepaGripperAxisX.setPositions[3].position+"Unit1.Em7.Config".cmSepaClampnCutterAxisX.setPositions[1].position;
   "Unit1.Em7.Config".cmSepaClampnCutterAxisX.setPositions[2].velocity := "Unit1.Em7.Config".cmSepaGripperAxisX.setPositions[3].velocity;
   "Unit1.Em7.Config".cmSepaClampnCutterAxisX.setPositions[2].acceleration := "Unit1.Em7.Config".cmSepaGripperAxisX.setPositions[3].acceleration;
   "Unit1.Em7.Config".cmSepaClampnCutterAxisX.setPositions[2].deceleration := "Unit1.Em7.Config".cmSepaGripperAxisX.setPositions[3].deceleration;
END_REGION

REGION Network 13: ******************** Equipment Control ********************
END_REGION

REGION Network 14: Interlink EM to Unit
   // This block links and unlinks the EM from the unit. The command to link/unlink can be set directly by the inputs of the block (e.g. to link/unlink based on any program logic) or through the InOut "hmiInterface". The block changes the output "isLinked" to true/false, depending on the command and if a change is allowed. A changed is allowed if the unit is in state aborted, clearing or stopped. The output "isLinked" is send back to the unit. If the EM is not linked, the unit ignores this EM.
   RUNG wire#powerrail
      "LUC_InterlinkToParent"(link := false, unlink := false, currentState := #unitStatus.state, hmiInterface := "Unit1.Em7.HmiInterface".em.interlinkMode, isLinked => #emFeedback.isLinked)
   END_RUNG
   // the same network as SCL:
   "LUC_InterlinkToParent"(link := false,
                           unlink := false,
                           currentState := #unitStatus.state,
                           hmiInterface := "Unit1.Em7.HmiInterface".em.interlinkMode,
                           isLinked => #emFeedback.isLinked);
END_REGION

REGION Network 15: Control EM
   // When linked, unitStatus is fully applied to unitStatusUsed.
   // When not linked, only acknowledge and safetyReleased from the unitStatus are applied. A direct EM control by hmiInterface or localInterface is possible.
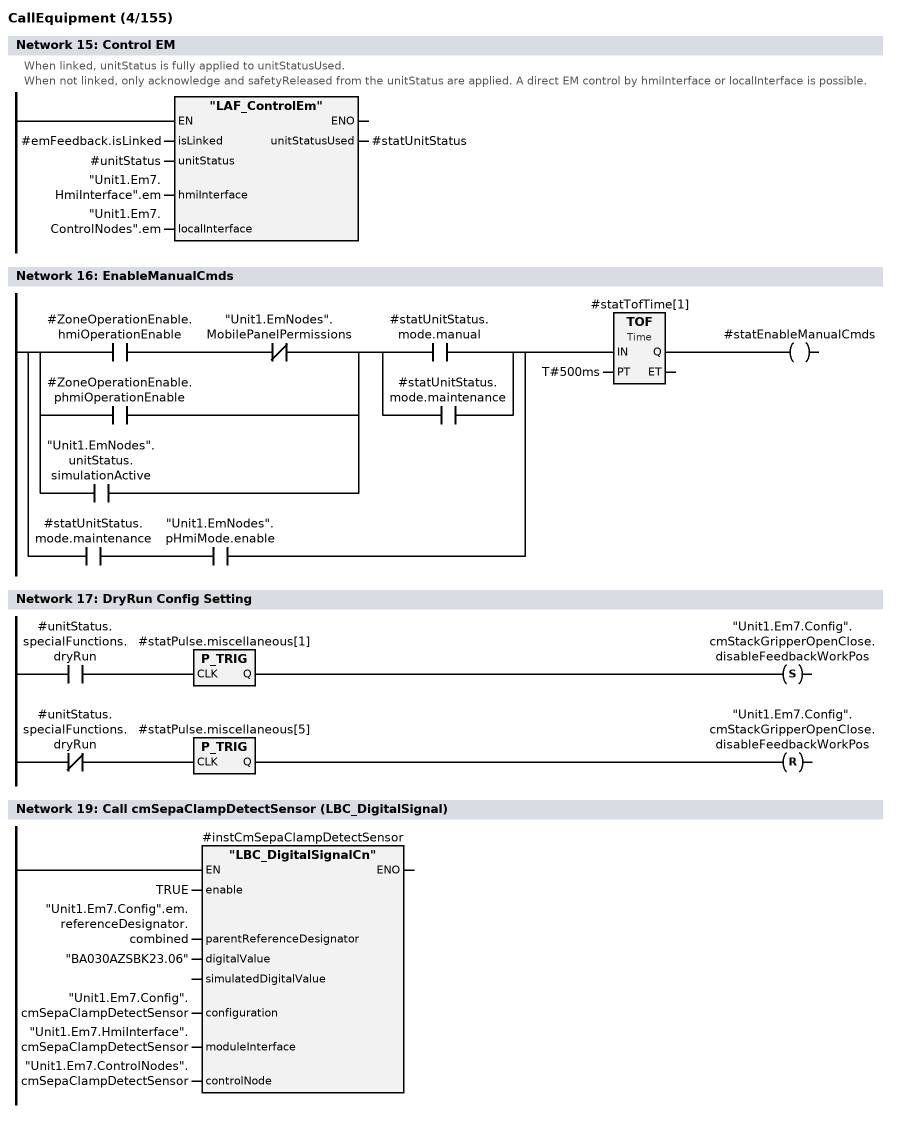
   RUNG wire#powerrail
      "LAF_ControlEm"(isLinked := #emFeedback.isLinked, unitStatus := #unitStatus, hmiInterface := "Unit1.Em7.HmiInterface".em, localInterface := "Unit1.Em7.ControlNodes".em, unitStatusUsed => #statUnitStatus)
   END_RUNG
   // the same network as SCL:
   "LAF_ControlEm"(isLinked := #emFeedback.isLinked,
                   unitStatus := #unitStatus,
                   hmiInterface := "Unit1.Em7.HmiInterface".em,
                   localInterface := "Unit1.Em7.ControlNodes".em,
                   unitStatusUsed => #statUnitStatus);
END_REGION

REGION Network 16: EnableManualCmds
   RUNG wire#powerrail
      Contact( #ZoneOperationEnable.hmiOperationEnable )
      I_Contact( "Unit1.EmNodes".MobilePanelPermissions )
      wire#w1
      Contact( #statUnitStatus.mode.manual )
      wire#w2
      { S7_Templates := "time_type := Time" } #statTofTime[1].TOF(pt := T#500ms, et =>)
      Coil( #statEnableManualCmds )
   END_RUNG
   RUNG wire#powerrail
      Contact( #ZoneOperationEnable.phmiOperationEnable )
   END_RUNG wire#w1
   RUNG wire#powerrail
      Contact( "Unit1.EmNodes".unitStatus.simulationActive )
   END_RUNG wire#w1
   RUNG wire#w1
      Contact( #statUnitStatus.mode.maintenance )
   END_RUNG wire#w2
   RUNG wire#powerrail
      Contact( #statUnitStatus.mode.maintenance )
      Contact( "Unit1.EmNodes".pHmiMode.enable )
   END_RUNG wire#w2
   // the same network as SCL:
   #statTofTime[1].TOF(IN := (((#ZoneOperationEnable.hmiOperationEnable AND NOT "Unit1.EmNodes".MobilePanelPermissions) OR #ZoneOperationEnable.phmiOperationEnable OR "Unit1.EmNodes".unitStatus.simulationActive) AND (#statUnitStatus.mode.manual OR #statUnitStatus.mode.maintenance)) OR (#statUnitStatus.mode.maintenance AND "Unit1.EmNodes".pHmiMode.enable),
                       PT := T#500ms);
   #statEnableManualCmds := #statTofTime[1].Q;
END_REGION

REGION Network 17: DryRun Config Setting
   RUNG wire#powerrail
      Contact( #unitStatus.specialFunctions.dryRun )
      P_Trig( #statPulse.miscellaneous[1] )
      S_Coil( "Unit1.Em7.Config".cmStackGripperOpenClose.disableFeedbackWorkPos )
   END_RUNG
   RUNG wire#powerrail
      I_Contact( #unitStatus.specialFunctions.dryRun )
      P_Trig( #statPulse.miscellaneous[5] )
      R_Coil( "Unit1.Em7.Config".cmStackGripperOpenClose.disableFeedbackWorkPos )
   END_RUNG
   // the same network as SCL:
   #_w1 := #unitStatus.specialFunctions.dryRun AND NOT #statPulse.miscellaneous[1];   // rising edge
   #statPulse.miscellaneous[1] := #unitStatus.specialFunctions.dryRun;
   IF #_w1 THEN "Unit1.Em7.Config".cmStackGripperOpenClose.disableFeedbackWorkPos := TRUE; END_IF;
   #_w2 := NOT #unitStatus.specialFunctions.dryRun AND NOT #statPulse.miscellaneous[5];   // rising edge
   #statPulse.miscellaneous[5] := NOT #unitStatus.specialFunctions.dryRun;
   IF #_w2 THEN "Unit1.Em7.Config".cmStackGripperOpenClose.disableFeedbackWorkPos := FALSE; END_IF;
END_REGION

REGION Network 18: ********** Control Modules (Sensors) **********
   // Call control modules that are sensors before the em logic (jobs and sequence), so that the latest value is used in the logic.
END_REGION

REGION Network 19: Call cmSepaClampDetectSensor (LBC_DigitalSignal)
   RUNG wire#powerrail
      #instCmSepaClampDetectSensor(enable := TRUE, parentReferenceDesignator := "Unit1.Em7.Config".em.referenceDesignator.combined, digitalValue := "BA030AZSBK23.06", simulatedDigitalValue :=, configuration := "Unit1.Em7.Config".cmSepaClampDetectSensor, moduleInterface := "Unit1.Em7.HmiInterface".cmSepaClampDetectSensor, controlNode := "Unit1.Em7.ControlNodes".cmSepaClampDetectSensor)
   END_RUNG
   // the same network as SCL:
   #instCmSepaClampDetectSensor(enable := TRUE,   // "LBC_DigitalSignalCn"
                           parentReferenceDesignator := "Unit1.Em7.Config".em.referenceDesignator.combined,
                           digitalValue := "BA030AZSBK23.06",
                           configuration := "Unit1.Em7.Config".cmSepaClampDetectSensor,
                           moduleInterface := "Unit1.Em7.HmiInterface".cmSepaClampDetectSensor,
                           controlNode := "Unit1.Em7.ControlNodes".cmSepaClampDetectSensor);
END_REGION

REGION Network 20: Call cmSepaGripperDetectSensor (LBC_DigitalSignal)
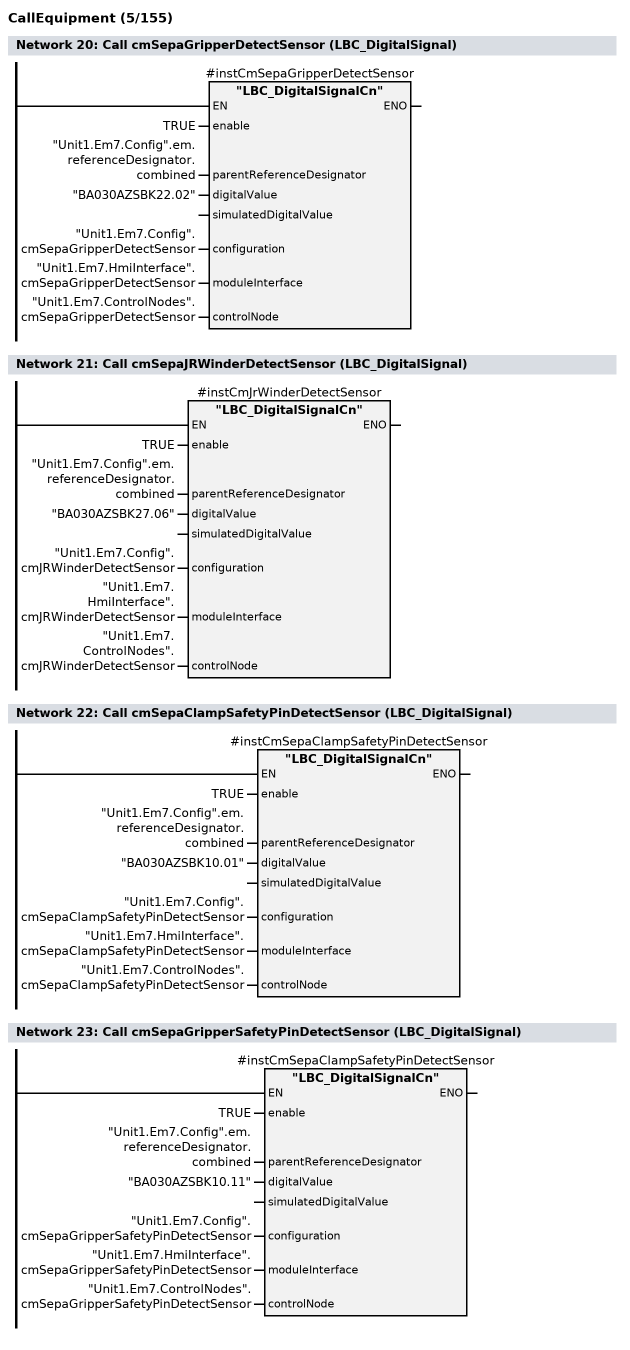
   RUNG wire#powerrail
      #instCmSepaGripperDetectSensor(enable := TRUE, parentReferenceDesignator := "Unit1.Em7.Config".em.referenceDesignator.combined, digitalValue := "BA030AZSBK22.02", simulatedDigitalValue :=, configuration := "Unit1.Em7.Config".cmSepaGripperDetectSensor, moduleInterface := "Unit1.Em7.HmiInterface".cmSepaGripperDetectSensor, controlNode := "Unit1.Em7.ControlNodes".cmSepaGripperDetectSensor)
   END_RUNG
   // the same network as SCL:
   #instCmSepaGripperDetectSensor(enable := TRUE,   // "LBC_DigitalSignalCn"
                           parentReferenceDesignator := "Unit1.Em7.Config".em.referenceDesignator.combined,
                           digitalValue := "BA030AZSBK22.02",
                           configuration := "Unit1.Em7.Config".cmSepaGripperDetectSensor,
                           moduleInterface := "Unit1.Em7.HmiInterface".cmSepaGripperDetectSensor,
                           controlNode := "Unit1.Em7.ControlNodes".cmSepaGripperDetectSensor);
END_REGION

REGION Network 21: Call cmSepaJRWinderDetectSensor (LBC_DigitalSignal)
   RUNG wire#powerrail
      #instCmJrWinderDetectSensor(enable := TRUE, parentReferenceDesignator := "Unit1.Em7.Config".em.referenceDesignator.combined, digitalValue := "BA030AZSBK27.06", simulatedDigitalValue :=, configuration := "Unit1.Em7.Config".cmJRWinderDetectSensor, moduleInterface := "Unit1.Em7.HmiInterface".cmJRWinderDetectSensor, controlNode := "Unit1.Em7.ControlNodes".cmJRWinderDetectSensor)
   END_RUNG
   // the same network as SCL:
   #instCmJrWinderDetectSensor(enable := TRUE,   // "LBC_DigitalSignalCn"
                           parentReferenceDesignator := "Unit1.Em7.Config".em.referenceDesignator.combined,
                           digitalValue := "BA030AZSBK27.06",
                           configuration := "Unit1.Em7.Config".cmJRWinderDetectSensor,
                           moduleInterface := "Unit1.Em7.HmiInterface".cmJRWinderDetectSensor,
                           controlNode := "Unit1.Em7.ControlNodes".cmJRWinderDetectSensor);
END_REGION

REGION Network 22: Call cmSepaClampSafetyPinDetectSensor (LBC_DigitalSignal)
   RUNG wire#powerrail
      #instCmSepaClampSafetyPinDetectSensor(enable := TRUE, parentReferenceDesignator := "Unit1.Em7.Config".em.referenceDesignator.combined, digitalValue := "BA030AZSBK10.01", simulatedDigitalValue :=, configuration := "Unit1.Em7.Config".cmSepaClampSafetyPinDetectSensor, moduleInterface := "Unit1.Em7.HmiInterface".cmSepaClampSafetyPinDetectSensor, controlNode := "Unit1.Em7.ControlNodes".cmSepaClampSafetyPinDetectSensor)
   END_RUNG
   // the same network as SCL:
   #instCmSepaClampSafetyPinDetectSensor(enable := TRUE,   // "LBC_DigitalSignalCn"
                           parentReferenceDesignator := "Unit1.Em7.Config".em.referenceDesignator.combined,
                           digitalValue := "BA030AZSBK10.01",
                           configuration := "Unit1.Em7.Config".cmSepaClampSafetyPinDetectSensor,
                           moduleInterface := "Unit1.Em7.HmiInterface".cmSepaClampSafetyPinDetectSensor,
                           controlNode := "Unit1.Em7.ControlNodes".cmSepaClampSafetyPinDetectSensor);
END_REGION

REGION Network 23: Call cmSepaGripperSafetyPinDetectSensor (LBC_DigitalSignal)
   RUNG wire#powerrail
      #instCmSepaClampSafetyPinDetectSensor(enable := TRUE, parentReferenceDesignator := "Unit1.Em7.Config".em.referenceDesignator.combined, digitalValue := "BA030AZSBK10.11", simulatedDigitalValue :=, configuration := "Unit1.Em7.Config".cmSepaGripperSafetyPinDetectSensor, moduleInterface := "Unit1.Em7.HmiInterface".cmSepaGripperSafetyPinDetectSensor, controlNode := "Unit1.Em7.ControlNodes".cmSepaGripperSafetyPinDetectSensor)
   END_RUNG
   // the same network as SCL:
   #instCmSepaClampSafetyPinDetectSensor(enable := TRUE,   // "LBC_DigitalSignalCn"
                           parentReferenceDesignator := "Unit1.Em7.Config".em.referenceDesignator.combined,
                           digitalValue := "BA030AZSBK10.11",
                           configuration := "Unit1.Em7.Config".cmSepaGripperSafetyPinDetectSensor,
                           moduleInterface := "Unit1.Em7.HmiInterface".cmSepaGripperSafetyPinDetectSensor,
                           controlNode := "Unit1.Em7.ControlNodes".cmSepaGripperSafetyPinDetectSensor);
END_REGION

REGION Network 24: ********** Equipment Logic **********
END_REGION

REGION Network 25: Map Unit Status to Sequence Status [1] Sepa Clamp
   // This block maps the unit status to the seuqnce status. Thus, it controls the sequence depending on the unit status. E.g. it sets the sequence to automatic when the unit state is in productions. This blocks work perfectly with the sequences provided in the AF. 
   // This typed block (MapUnitStatusToSequence) could be adjusted to specific application requirements or if other, user-defined sequences are used.
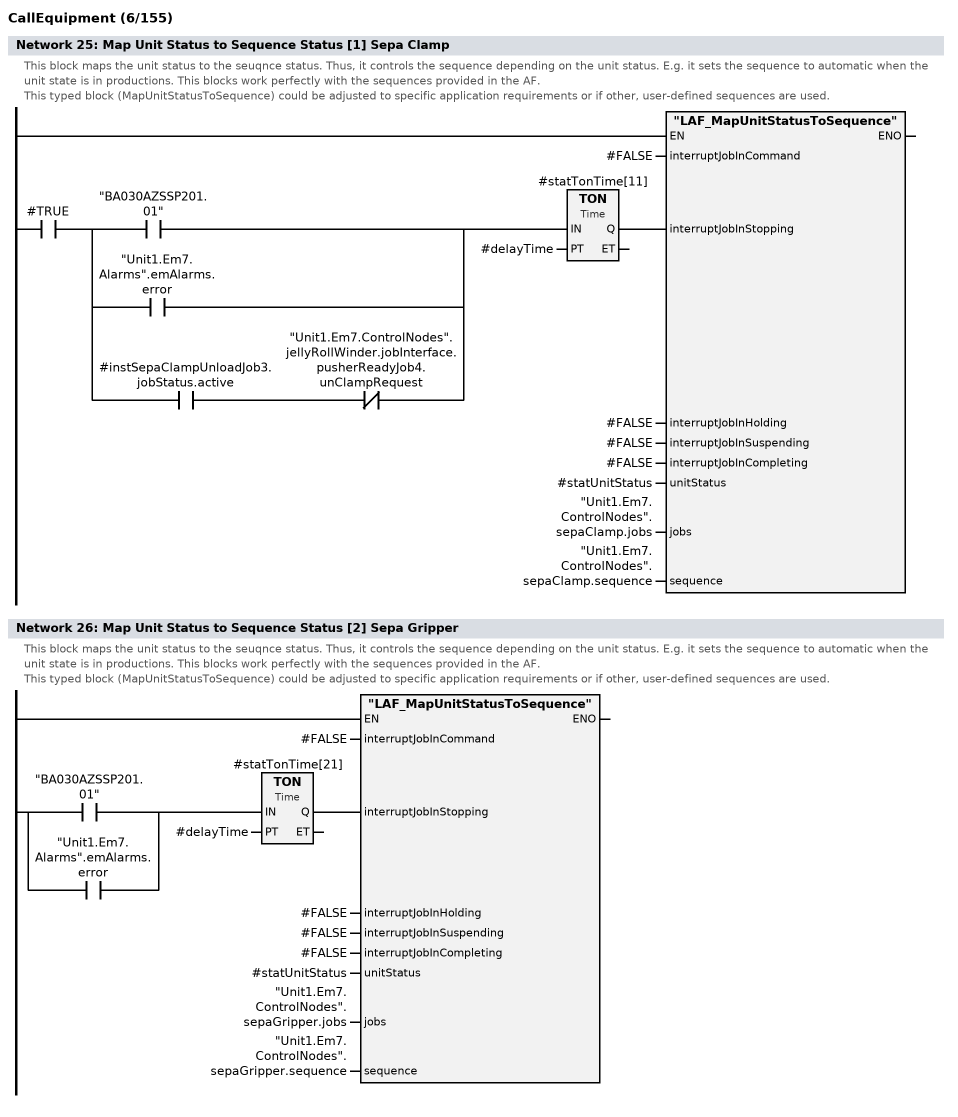
   RUNG wire#powerrail
      "LAF_MapUnitStatusToSequence"(interruptJobInStopping := wire#w3, interruptJobInCommand := #FALSE, interruptJobInHolding := #FALSE, interruptJobInSuspending := #FALSE, interruptJobInCompleting := #FALSE, unitStatus := #statUnitStatus, jobs := "Unit1.Em7.ControlNodes".sepaClamp.jobs, sequence := "Unit1.Em7.ControlNodes".sepaClamp.sequence)
   END_RUNG
   RUNG wire#powerrail
      Contact( #TRUE )
      wire#w1
      Contact( "BA030AZSSP201.01" )
      wire#w2
      { S7_Templates := "time_type := Time" } #statTonTime[11].TON(pt := #delayTime, et =>)
   END_RUNG wire#w3
   RUNG wire#w1
      Contact( "Unit1.Em7.Alarms".emAlarms.error )
   END_RUNG wire#w2
   RUNG wire#w1
      Contact( #instSepaClampUnloadJob3.jobStatus.active )
      I_Contact( "Unit1.Em7.ControlNodes".jellyRollWinder.jobInterface.pusherReadyJob4.unClampRequest )
   END_RUNG wire#w2
   // the same network as SCL:
   #statTonTime[11].TON(IN := #TRUE AND ("BA030AZSSP201.01" OR "Unit1.Em7.Alarms".emAlarms.error OR (#instSepaClampUnloadJob3.jobStatus.active AND NOT "Unit1.Em7.ControlNodes".jellyRollWinder.jobInterface.pusherReadyJob4.unClampRequest)),
                        PT := #delayTime);
   "LAF_MapUnitStatusToSequence"(interruptJobInCommand := #FALSE,
                           interruptJobInStopping := #statTonTime[11].Q,
                           interruptJobInHolding := #FALSE,
                           interruptJobInSuspending := #FALSE,
                           interruptJobInCompleting := #FALSE,
                           unitStatus := #statUnitStatus,
                           jobs := "Unit1.Em7.ControlNodes".sepaClamp.jobs,
                           sequence := "Unit1.Em7.ControlNodes".sepaClamp.sequence);
END_REGION

REGION Network 26: Map Unit Status to Sequence Status [2] Sepa Gripper
   // This block maps the unit status to the seuqnce status. Thus, it controls the sequence depending on the unit status. E.g. it sets the sequence to automatic when the unit state is in productions. This blocks work perfectly with the sequences provided in the AF. 
   // This typed block (MapUnitStatusToSequence) could be adjusted to specific application requirements or if other, user-defined sequences are used.
   RUNG wire#powerrail
      "LAF_MapUnitStatusToSequence"(interruptJobInStopping := wire#w2, interruptJobInCommand := #FALSE, interruptJobInHolding := #FALSE, interruptJobInSuspending := #FALSE, interruptJobInCompleting := #FALSE, unitStatus := #statUnitStatus, jobs := "Unit1.Em7.ControlNodes".sepaGripper.jobs, sequence := "Unit1.Em7.ControlNodes".sepaGripper.sequence)
   END_RUNG
   RUNG wire#powerrail
      Contact( "BA030AZSSP201.01" )
      wire#w1
      { S7_Templates := "time_type := Time" } #statTonTime[21].TON(pt := #delayTime, et =>)
   END_RUNG wire#w2
   RUNG wire#powerrail
      Contact( "Unit1.Em7.Alarms".emAlarms.error )
   END_RUNG wire#w1
   // the same network as SCL:
   #statTonTime[21].TON(IN := "BA030AZSSP201.01" OR "Unit1.Em7.Alarms".emAlarms.error, PT := #delayTime);
   "LAF_MapUnitStatusToSequence"(interruptJobInCommand := #FALSE,
                           interruptJobInStopping := #statTonTime[21].Q,
                           interruptJobInHolding := #FALSE,
                           interruptJobInSuspending := #FALSE,
                           interruptJobInCompleting := #FALSE,
                           unitStatus := #statUnitStatus,
                           jobs := "Unit1.Em7.ControlNodes".sepaGripper.jobs,
                           sequence := "Unit1.Em7.ControlNodes".sepaGripper.sequence);
END_REGION

REGION Network 27: Map Unit Status to Sequence Status [3] Jelly Roll Winder
   // This block maps the unit status to the seuqnce status. Thus, it controls the sequence depending on the unit status. E.g. it sets the sequence to automatic when the unit state is in productions. This blocks work perfectly with the sequences provided in the AF. 
   // This typed block (MapUnitStatusToSequence) could be adjusted to specific application requirements or if other, user-defined sequences are used.
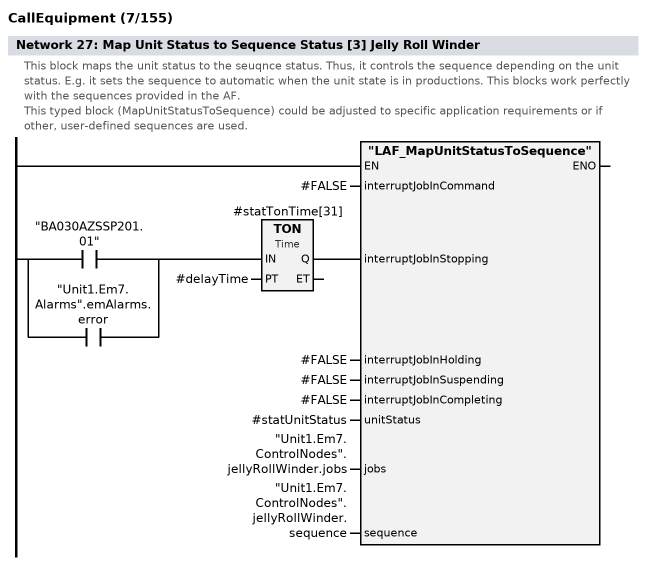
   RUNG wire#powerrail
      "LAF_MapUnitStatusToSequence"(interruptJobInStopping := wire#w2, interruptJobInCommand := #FALSE, interruptJobInHolding := #FALSE, interruptJobInSuspending := #FALSE, interruptJobInCompleting := #FALSE, unitStatus := #statUnitStatus, jobs := "Unit1.Em7.ControlNodes".jellyRollWinder.jobs, sequence := "Unit1.Em7.ControlNodes".jellyRollWinder.sequence)
   END_RUNG
   RUNG wire#powerrail
      Contact( "BA030AZSSP201.01" )
      wire#w1
      { S7_Templates := "time_type := Time" } #statTonTime[31].TON(pt := #delayTime, et =>)
   END_RUNG wire#w2
   RUNG wire#powerrail
      Contact( "Unit1.Em7.Alarms".emAlarms.error )
   END_RUNG wire#w1
   // the same network as SCL:
   #statTonTime[31].TON(IN := "BA030AZSSP201.01" OR "Unit1.Em7.Alarms".emAlarms.error, PT := #delayTime);
   "LAF_MapUnitStatusToSequence"(interruptJobInCommand := #FALSE,
                           interruptJobInStopping := #statTonTime[31].Q,
                           interruptJobInHolding := #FALSE,
                           interruptJobInSuspending := #FALSE,
                           interruptJobInCompleting := #FALSE,
                           unitStatus := #statUnitStatus,
                           jobs := "Unit1.Em7.ControlNodes".jellyRollWinder.jobs,
                           sequence := "Unit1.Em7.ControlNodes".jellyRollWinder.sequence);
END_REGION

REGION Network 29: Sepa Clamp Select Job
   // Decide which Step Sequence to start depending on the OMAC State and EM conditions
   // First Move Block is to Initialize the jobSelect Number
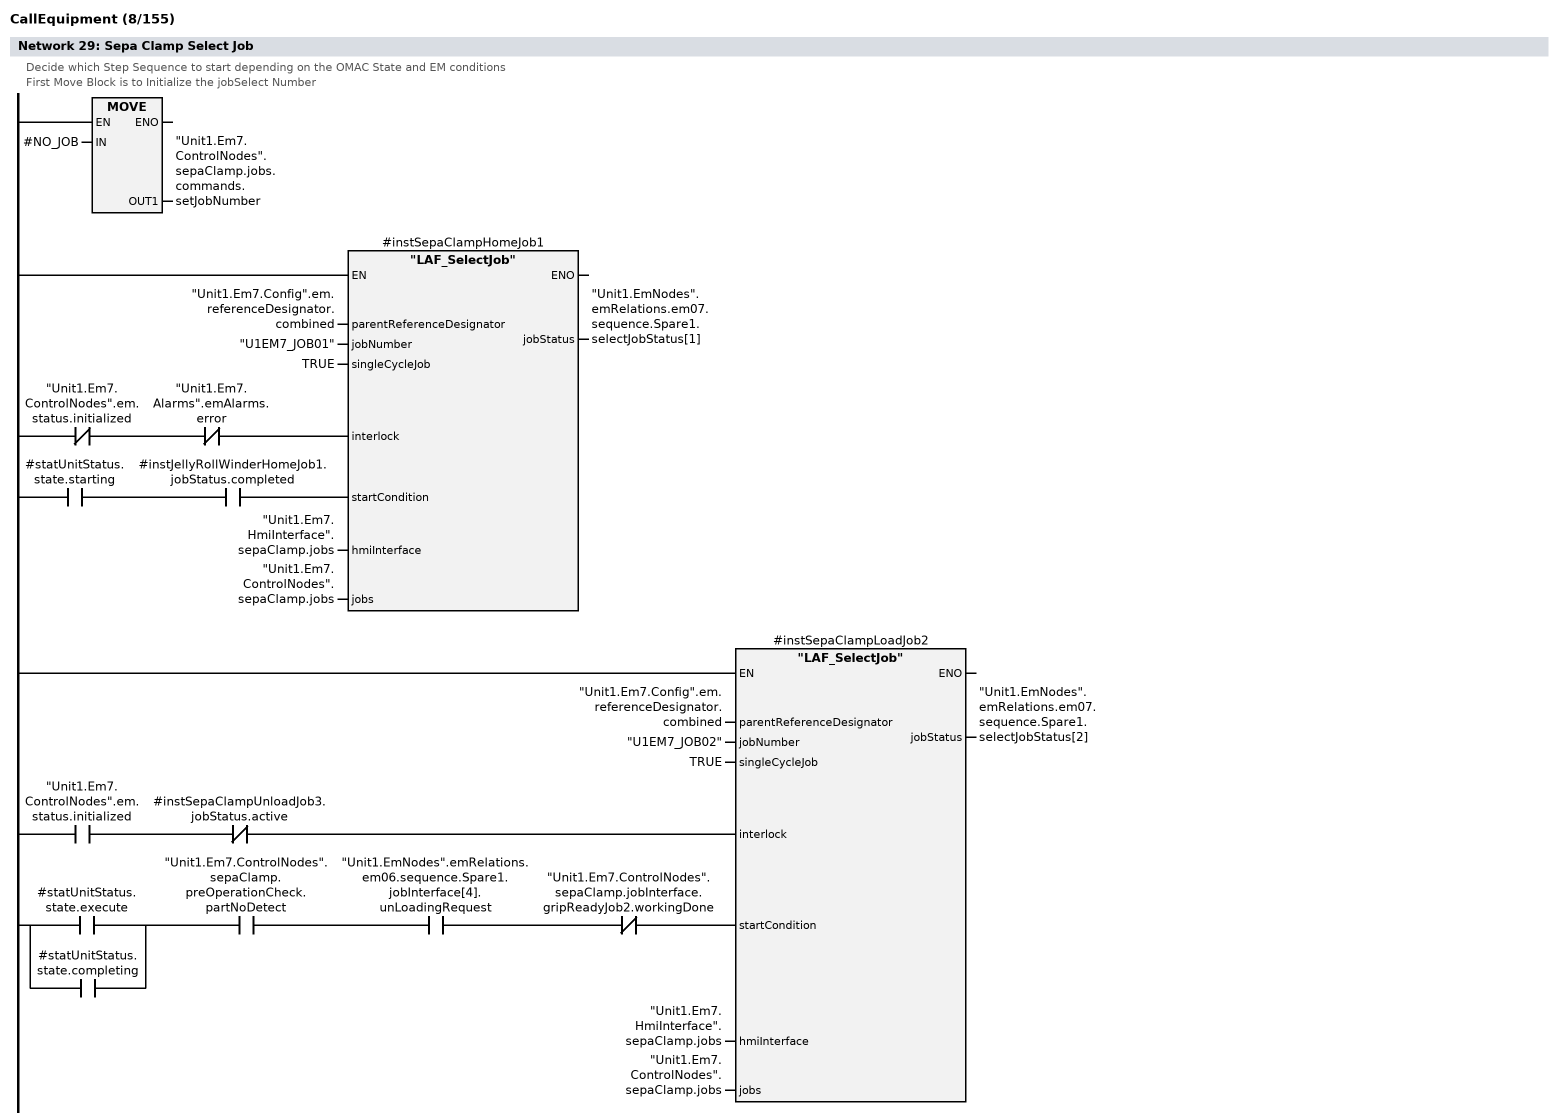
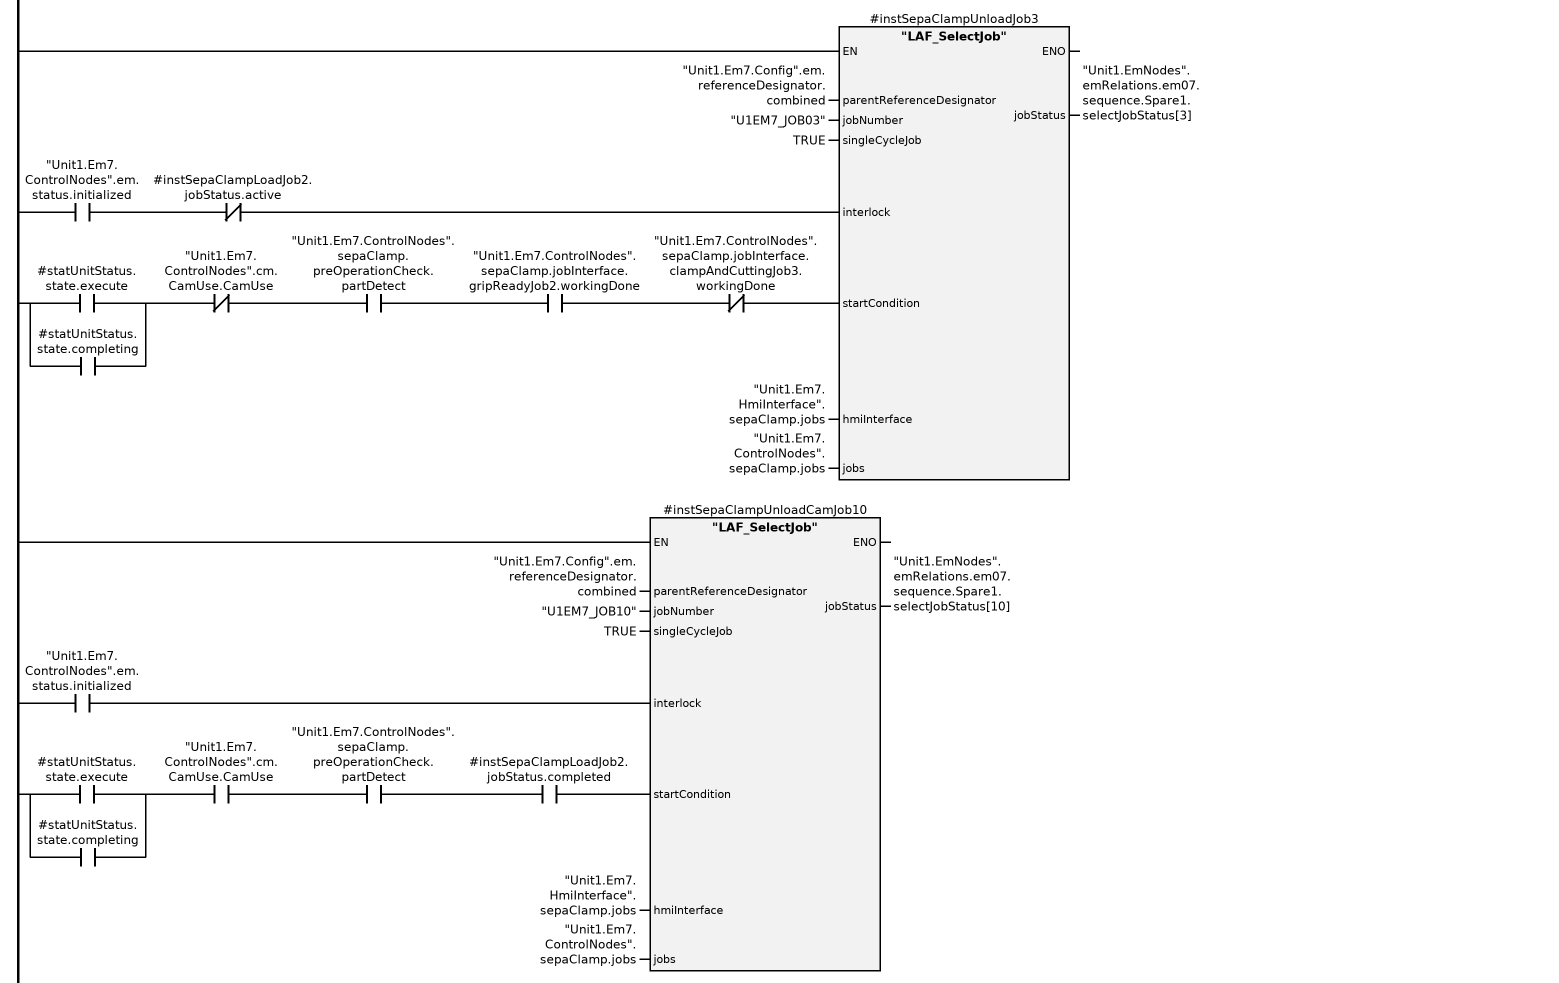
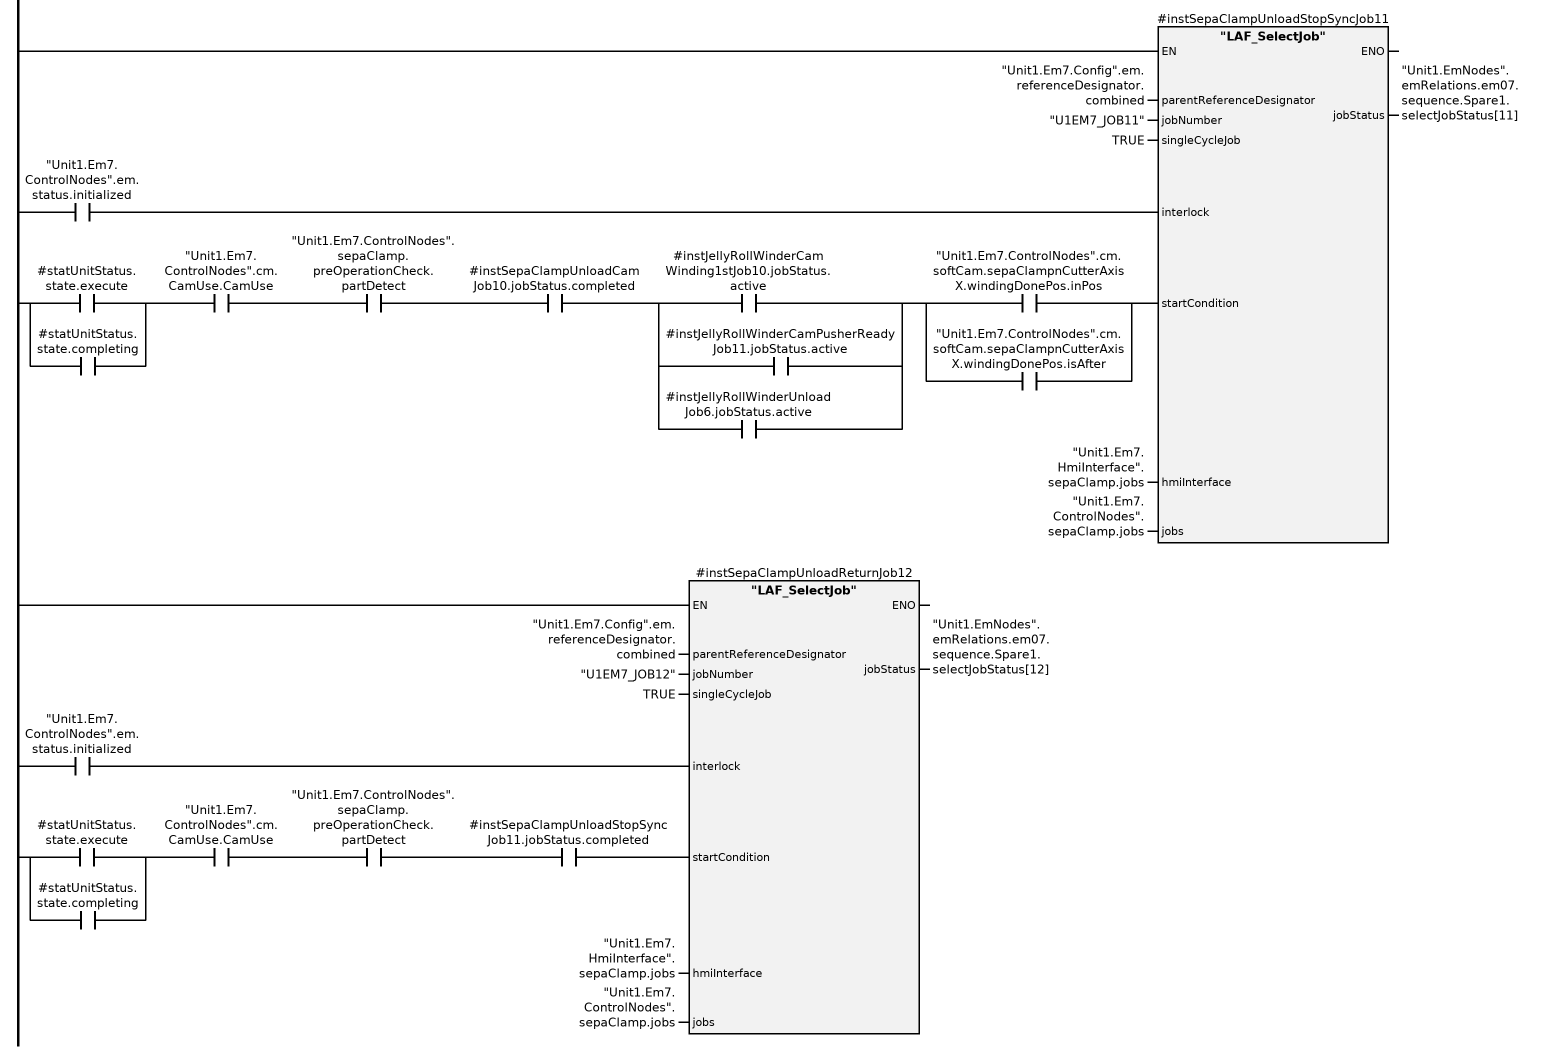
   RUNG wire#powerrail
      Move(in := #NO_JOB, out1 => "Unit1.Em7.ControlNodes".sepaClamp.jobs.commands.setJobNumber)
   END_RUNG
   RUNG wire#powerrail
      #instSepaClampHomeJob1(interlock := wire#w1, startCondition := wire#w2, parentReferenceDesignator := "Unit1.Em7.Config".em.referenceDesignator.combined, jobNumber := "U1EM7_JOB01", singleCycleJob := TRUE, hmiInterface := "Unit1.Em7.HmiInterface".sepaClamp.jobs, jobs := "Unit1.Em7.ControlNodes".sepaClamp.jobs, jobStatus => "Unit1.EmNodes".emRelations.em07.sequence.Spare1.selectJobStatus[1])
   END_RUNG
   RUNG wire#powerrail
      I_Contact( "Unit1.Em7.ControlNodes".em.status.initialized )
      I_Contact( "Unit1.Em7.Alarms".emAlarms.error )
   END_RUNG wire#w1
   RUNG wire#powerrail
      Contact( #statUnitStatus.state.starting )
      Contact( #instJellyRollWinderHomeJob1.jobStatus.completed )
   END_RUNG wire#w2
   RUNG wire#powerrail
      #instSepaClampLoadJob2(interlock := wire#w3, startCondition := wire#w5, parentReferenceDesignator := "Unit1.Em7.Config".em.referenceDesignator.combined, jobNumber := "U1EM7_JOB02", singleCycleJob := TRUE, hmiInterface := "Unit1.Em7.HmiInterface".sepaClamp.jobs, jobs := "Unit1.Em7.ControlNodes".sepaClamp.jobs, jobStatus => "Unit1.EmNodes".emRelations.em07.sequence.Spare1.selectJobStatus[2])
   END_RUNG
   RUNG wire#powerrail
      Contact( "Unit1.Em7.ControlNodes".em.status.initialized )
      I_Contact( #instSepaClampUnloadJob3.jobStatus.active )
   END_RUNG wire#w3
   RUNG wire#powerrail
      Contact( #statUnitStatus.state.execute )
      wire#w4
      Contact( "Unit1.Em7.ControlNodes".sepaClamp.preOperationCheck.partNoDetect )
      Contact( "Unit1.EmNodes".emRelations.em06.sequence.Spare1.jobInterface[4].unLoadingRequest )
      I_Contact( "Unit1.Em7.ControlNodes".sepaClamp.jobInterface.gripReadyJob2.workingDone )
   END_RUNG wire#w5
   RUNG wire#powerrail
      Contact( #statUnitStatus.state.completing )
   END_RUNG wire#w4
   RUNG wire#powerrail
      #instSepaClampUnloadJob3(interlock := wire#w6, startCondition := wire#w8, parentReferenceDesignator := "Unit1.Em7.Config".em.referenceDesignator.combined, jobNumber := "U1EM7_JOB03", singleCycleJob := TRUE, hmiInterface := "Unit1.Em7.HmiInterface".sepaClamp.jobs, jobs := "Unit1.Em7.ControlNodes".sepaClamp.jobs, jobStatus => "Unit1.EmNodes".emRelations.em07.sequence.Spare1.selectJobStatus[3])
   END_RUNG
   RUNG wire#powerrail
      Contact( "Unit1.Em7.ControlNodes".em.status.initialized )
      I_Contact( #instSepaClampLoadJob2.jobStatus.active )
   END_RUNG wire#w6
   RUNG wire#powerrail
      Contact( #statUnitStatus.state.execute )
      wire#w7
      I_Contact( "Unit1.Em7.ControlNodes".cm.CamUse.CamUse )
      Contact( "Unit1.Em7.ControlNodes".sepaClamp.preOperationCheck.partDetect )
      Contact( "Unit1.Em7.ControlNodes".sepaClamp.jobInterface.gripReadyJob2.workingDone )
      I_Contact( "Unit1.Em7.ControlNodes".sepaClamp.jobInterface.clampAndCuttingJob3.workingDone )
   END_RUNG wire#w8
   RUNG wire#powerrail
      Contact( #statUnitStatus.state.completing )
   END_RUNG wire#w7
   RUNG wire#powerrail
      #instSepaClampUnloadCamJob10(interlock := wire#w9, startCondition := wire#w11, parentReferenceDesignator := "Unit1.Em7.Config".em.referenceDesignator.combined, jobNumber := "U1EM7_JOB10", singleCycleJob := TRUE, hmiInterface := "Unit1.Em7.HmiInterface".sepaClamp.jobs, jobs := "Unit1.Em7.ControlNodes".sepaClamp.jobs, jobStatus => "Unit1.EmNodes".emRelations.em07.sequence.Spare1.selectJobStatus[10])
   END_RUNG
   RUNG wire#powerrail
      Contact( "Unit1.Em7.ControlNodes".em.status.initialized )
   END_RUNG wire#w9
   RUNG wire#powerrail
      Contact( #statUnitStatus.state.execute )
      wire#w10
      Contact( "Unit1.Em7.ControlNodes".cm.CamUse.CamUse )
      Contact( "Unit1.Em7.ControlNodes".sepaClamp.preOperationCheck.partDetect )
      Contact( #instSepaClampLoadJob2.jobStatus.completed )
   END_RUNG wire#w11
   RUNG wire#powerrail
      Contact( #statUnitStatus.state.completing )
   END_RUNG wire#w10
   RUNG wire#powerrail
      #instSepaClampUnloadStopSyncJob11(interlock := wire#w12, startCondition := wire#w16, parentReferenceDesignator := "Unit1.Em7.Config".em.referenceDesignator.combined, jobNumber := "U1EM7_JOB11", singleCycleJob := TRUE, hmiInterface := "Unit1.Em7.HmiInterface".sepaClamp.jobs, jobs := "Unit1.Em7.ControlNodes".sepaClamp.jobs, jobStatus => "Unit1.EmNodes".emRelations.em07.sequence.Spare1.selectJobStatus[11])
   END_RUNG
   RUNG wire#powerrail
      Contact( "Unit1.Em7.ControlNodes".em.status.initialized )
   END_RUNG wire#w12
   RUNG wire#powerrail
      Contact( #statUnitStatus.state.execute )
      wire#w13
      Contact( "Unit1.Em7.ControlNodes".cm.CamUse.CamUse )
      Contact( "Unit1.Em7.ControlNodes".sepaClamp.preOperationCheck.partDetect )
      Contact( #instSepaClampUnloadCamJob10.jobStatus.completed )
      wire#w14
      Contact( #instJellyRollWinderCamWinding1stJob10.jobStatus.active )
      wire#w15
      Contact( "Unit1.Em7.ControlNodes".cm.softCam.sepaClampnCutterAxisX.windingDonePos.inPos )
   END_RUNG wire#w16
   RUNG wire#powerrail
      Contact( #statUnitStatus.state.completing )
   END_RUNG wire#w13
   RUNG wire#w14
      Contact( #instJellyRollWinderCamPusherReadyJob11.jobStatus.active )
   END_RUNG wire#w15
   RUNG wire#w14
      Contact( #instJellyRollWinderUnloadJob6.jobStatus.active )
   END_RUNG wire#w15
   RUNG wire#w15
      Contact( "Unit1.Em7.ControlNodes".cm.softCam.sepaClampnCutterAxisX.windingDonePos.isAfter )
   END_RUNG wire#w16
   RUNG wire#powerrail
      #instSepaClampUnloadReturnJob12(interlock := wire#w17, startCondition := wire#w19, parentReferenceDesignator := "Unit1.Em7.Config".em.referenceDesignator.combined, jobNumber := "U1EM7_JOB12", singleCycleJob := TRUE, hmiInterface := "Unit1.Em7.HmiInterface".sepaClamp.jobs, jobs := "Unit1.Em7.ControlNodes".sepaClamp.jobs, jobStatus => "Unit1.EmNodes".emRelations.em07.sequence.Spare1.selectJobStatus[12])
   END_RUNG
   RUNG wire#powerrail
      Contact( "Unit1.Em7.ControlNodes".em.status.initialized )
   END_RUNG wire#w17
   RUNG wire#powerrail
      Contact( #statUnitStatus.state.execute )
      wire#w18
      Contact( "Unit1.Em7.ControlNodes".cm.CamUse.CamUse )
      Contact( "Unit1.Em7.ControlNodes".sepaClamp.preOperationCheck.partDetect )
      Contact( #instSepaClampUnloadStopSyncJob11.jobStatus.completed )
   END_RUNG wire#w19
   RUNG wire#powerrail
      Contact( #statUnitStatus.state.completing )
   END_RUNG wire#w18
   // the same network as SCL:
   "Unit1.Em7.ControlNodes".sepaClamp.jobs.commands.setJobNumber := #NO_JOB;
   #instSepaClampHomeJob1(parentReferenceDesignator := "Unit1.Em7.Config".em.referenceDesignator.combined,   // "LAF_SelectJob"
                          jobNumber := "U1EM7_JOB01",
                          singleCycleJob := TRUE,
                          interlock := NOT "Unit1.Em7.ControlNodes".em.status.initialized AND NOT "Unit1.Em7.Alarms".emAlarms.error,
                          startCondition := #statUnitStatus.state.starting AND #instJellyRollWinderHomeJob1.jobStatus.completed,
                          hmiInterface := "Unit1.Em7.HmiInterface".sepaClamp.jobs,
                          jobs := "Unit1.Em7.ControlNodes".sepaClamp.jobs,
                          jobStatus => "Unit1.EmNodes".emRelations.em07.sequence.Spare1.selectJobStatus[1]);
   #instSepaClampLoadJob2(parentReferenceDesignator := "Unit1.Em7.Config".em.referenceDesignator.combined,   // "LAF_SelectJob"
                          jobNumber := "U1EM7_JOB02",
                          singleCycleJob := TRUE,
                          interlock := "Unit1.Em7.ControlNodes".em.status.initialized AND NOT #instSepaClampUnloadJob3.jobStatus.active,
                          startCondition := (#statUnitStatus.state.execute OR #statUnitStatus.state.completing) AND "Unit1.Em7.ControlNodes".sepaClamp.preOperationCheck.partNoDetect AND "Unit1.EmNodes".emRelations.em06.sequence.Spare1.jobInterface[4].unLoadingRequest AND NOT "Unit1.Em7.ControlNodes".sepaClamp.jobInterface.gripReadyJob2.workingDone,
                          hmiInterface := "Unit1.Em7.HmiInterface".sepaClamp.jobs,
                          jobs := "Unit1.Em7.ControlNodes".sepaClamp.jobs,
                          jobStatus => "Unit1.EmNodes".emRelations.em07.sequence.Spare1.selectJobStatus[2]);
   #instSepaClampUnloadJob3(parentReferenceDesignator := "Unit1.Em7.Config".em.referenceDesignator.combined,   // "LAF_SelectJob"
                           jobNumber := "U1EM7_JOB03",
                           singleCycleJob := TRUE,
                           interlock := "Unit1.Em7.ControlNodes".em.status.initialized AND NOT #instSepaClampLoadJob2.jobStatus.active,
                           startCondition := (#statUnitStatus.state.execute OR #statUnitStatus.state.completing) AND NOT "Unit1.Em7.ControlNodes".cm.CamUse.CamUse AND "Unit1.Em7.ControlNodes".sepaClamp.preOperationCheck.partDetect AND "Unit1.Em7.ControlNodes".sepaClamp.jobInterface.gripReadyJob2.workingDone AND NOT "Unit1.Em7.ControlNodes".sepaClamp.jobInterface.clampAndCuttingJob3.workingDone,
                           hmiInterface := "Unit1.Em7.HmiInterface".sepaClamp.jobs,
                           jobs := "Unit1.Em7.ControlNodes".sepaClamp.jobs,
                           jobStatus => "Unit1.EmNodes".emRelations.em07.sequence.Spare1.selectJobStatus[3]);
   #instSepaClampUnloadCamJob10(parentReferenceDesignator := "Unit1.Em7.Config".em.referenceDesignator.combined,   // "LAF_SelectJob"
                           jobNumber := "U1EM7_JOB10",
                           singleCycleJob := TRUE,
                           interlock := "Unit1.Em7.ControlNodes".em.status.initialized,
                           startCondition := (#statUnitStatus.state.execute OR #statUnitStatus.state.completing) AND "Unit1.Em7.ControlNodes".cm.CamUse.CamUse AND "Unit1.Em7.ControlNodes".sepaClamp.preOperationCheck.partDetect AND #instSepaClampLoadJob2.jobStatus.completed,
                           hmiInterface := "Unit1.Em7.HmiInterface".sepaClamp.jobs,
                           jobs := "Unit1.Em7.ControlNodes".sepaClamp.jobs,
                           jobStatus => "Unit1.EmNodes".emRelations.em07.sequence.Spare1.selectJobStatus[10]);
   #instSepaClampUnloadStopSyncJob11(parentReferenceDesignator := "Unit1.Em7.Config".em.referenceDesignator.combined,   // "LAF_SelectJob"
                           jobNumber := "U1EM7_JOB11",
                           singleCycleJob := TRUE,
                           interlock := "Unit1.Em7.ControlNodes".em.status.initialized,
                           startCondition := (#statUnitStatus.state.execute OR #statUnitStatus.state.completing) AND "Unit1.Em7.ControlNodes".cm.CamUse.CamUse AND "Unit1.Em7.ControlNodes".sepaClamp.preOperationCheck.partDetect AND #instSepaClampUnloadCamJob10.jobStatus.completed AND (#instJellyRollWinderCamWinding1stJob10.jobStatus.active OR #instJellyRollWinderCamPusherReadyJob11.jobStatus.active OR #instJellyRollWinderUnloadJob6.jobStatus.active) AND ("Unit1.Em7.ControlNodes".cm.softCam.sepaClampnCutterAxisX.windingDonePos.inPos OR "Unit1.Em7.ControlNodes".cm.softCam.sepaClampnCutterAxisX.windingDonePos.isAfter),
                           hmiInterface := "Unit1.Em7.HmiInterface".sepaClamp.jobs,
                           jobs := "Unit1.Em7.ControlNodes".sepaClamp.jobs,
                           jobStatus => "Unit1.EmNodes".emRelations.em07.sequence.Spare1.selectJobStatus[11]);
   #instSepaClampUnloadReturnJob12(parentReferenceDesignator := "Unit1.Em7.Config".em.referenceDesignator.combined,   // "LAF_SelectJob"
                           jobNumber := "U1EM7_JOB12",
                           singleCycleJob := TRUE,
                           interlock := "Unit1.Em7.ControlNodes".em.status.initialized,
                           startCondition := (#statUnitStatus.state.execute OR #statUnitStatus.state.completing) AND "Unit1.Em7.ControlNodes".cm.CamUse.CamUse AND "Unit1.Em7.ControlNodes".sepaClamp.preOperationCheck.partDetect AND #instSepaClampUnloadStopSyncJob11.jobStatus.completed,
                           hmiInterface := "Unit1.Em7.HmiInterface".sepaClamp.jobs,
                           jobs := "Unit1.Em7.ControlNodes".sepaClamp.jobs,
                           jobStatus => "Unit1.EmNodes".emRelations.em07.sequence.Spare1.selectJobStatus[12]);
END_REGION

REGION Network 30: Sepa Clamp Job Interface [Loading]
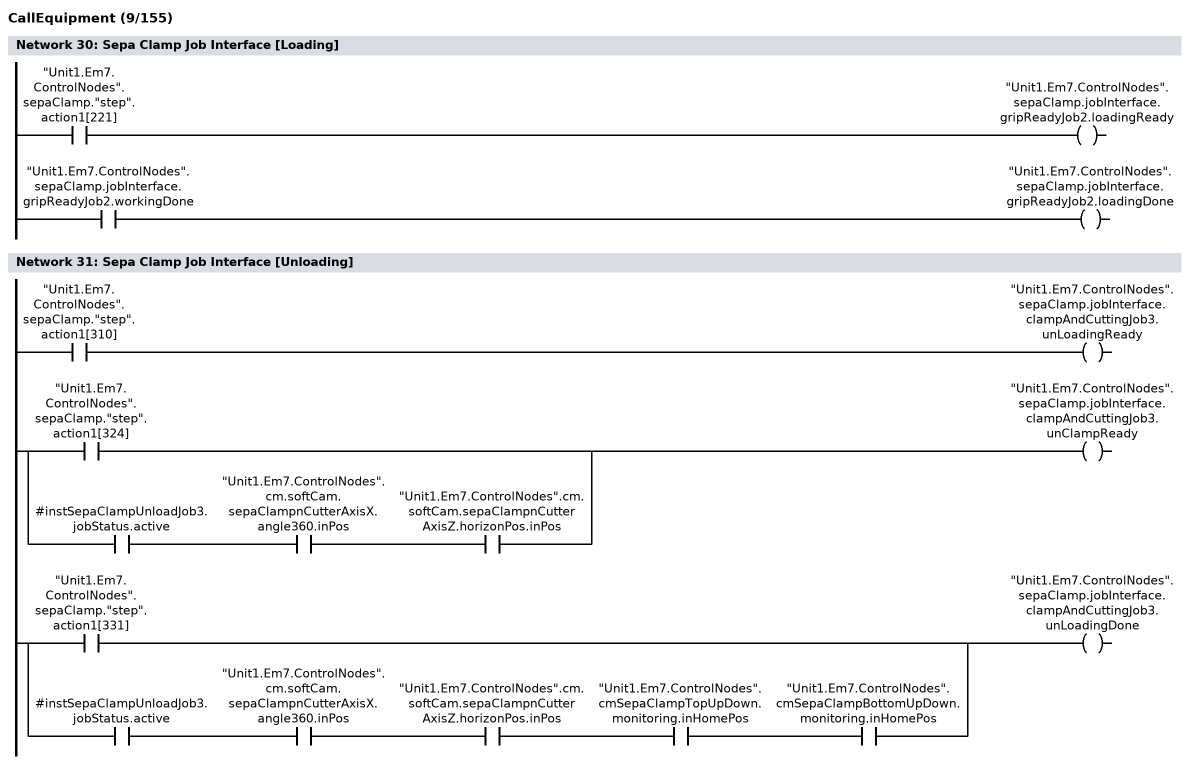
   RUNG wire#powerrail
      Contact( "Unit1.Em7.ControlNodes".sepaClamp."step".action1[221] )
      Coil( "Unit1.Em7.ControlNodes".sepaClamp.jobInterface.gripReadyJob2.loadingReady )
   END_RUNG
   RUNG wire#powerrail
      Contact( "Unit1.Em7.ControlNodes".sepaClamp.jobInterface.gripReadyJob2.workingDone )
      Coil( "Unit1.Em7.ControlNodes".sepaClamp.jobInterface.gripReadyJob2.loadingDone )
   END_RUNG
   // the same network as SCL:
   "Unit1.Em7.ControlNodes".sepaClamp.jobInterface.gripReadyJob2.loadingReady := "Unit1.Em7.ControlNodes".sepaClamp."step".action1[221];
   "Unit1.Em7.ControlNodes".sepaClamp.jobInterface.gripReadyJob2.loadingDone := "Unit1.Em7.ControlNodes".sepaClamp.jobInterface.gripReadyJob2.workingDone;
END_REGION

REGION Network 31: Sepa Clamp Job Interface [Unloading]
   RUNG wire#powerrail
      Contact( "Unit1.Em7.ControlNodes".sepaClamp."step".action1[310] )
      Coil( "Unit1.Em7.ControlNodes".sepaClamp.jobInterface.clampAndCuttingJob3.unLoadingReady )
   END_RUNG
   RUNG wire#powerrail
      Contact( "Unit1.Em7.ControlNodes".sepaClamp."step".action1[324] )
      wire#w1
      Coil( "Unit1.Em7.ControlNodes".sepaClamp.jobInterface.clampAndCuttingJob3.unClampReady )
   END_RUNG
   RUNG wire#powerrail
      Contact( #instSepaClampUnloadJob3.jobStatus.active )
      Contact( "Unit1.Em7.ControlNodes".cm.softCam.sepaClampnCutterAxisX.angle360.inPos )
      Contact( "Unit1.Em7.ControlNodes".cm.softCam.sepaClampnCutterAxisZ.horizonPos.inPos )
   END_RUNG wire#w1
   RUNG wire#powerrail
      Contact( "Unit1.Em7.ControlNodes".sepaClamp."step".action1[331] )
      wire#w2
      Coil( "Unit1.Em7.ControlNodes".sepaClamp.jobInterface.clampAndCuttingJob3.unLoadingDone )
   END_RUNG
   RUNG wire#powerrail
      Contact( #instSepaClampUnloadJob3.jobStatus.active )
      Contact( "Unit1.Em7.ControlNodes".cm.softCam.sepaClampnCutterAxisX.angle360.inPos )
      Contact( "Unit1.Em7.ControlNodes".cm.softCam.sepaClampnCutterAxisZ.horizonPos.inPos )
      Contact( "Unit1.Em7.ControlNodes".cmSepaClampTopUpDown.monitoring.inHomePos )
      Contact( "Unit1.Em7.ControlNodes".cmSepaClampBottomUpDown.monitoring.inHomePos )
   END_RUNG wire#w2
   // the same network as SCL:
   "Unit1.Em7.ControlNodes".sepaClamp.jobInterface.clampAndCuttingJob3.unLoadingReady := "Unit1.Em7.ControlNodes".sepaClamp."step".action1[310];
   "Unit1.Em7.ControlNodes".sepaClamp.jobInterface.clampAndCuttingJob3.unClampReady := "Unit1.Em7.ControlNodes".sepaClamp."step".action1[324] OR (#instSepaClampUnloadJob3.jobStatus.active AND "Unit1.Em7.ControlNodes".cm.softCam.sepaClampnCutterAxisX.angle360.inPos AND "Unit1.Em7.ControlNodes".cm.softCam.sepaClampnCutterAxisZ.horizonPos.inPos);
   "Unit1.Em7.ControlNodes".sepaClamp.jobInterface.clampAndCuttingJob3.unLoadingDone := "Unit1.Em7.ControlNodes".sepaClamp."step".action1[331] OR (#instSepaClampUnloadJob3.jobStatus.active AND "Unit1.Em7.ControlNodes".cm.softCam.sepaClampnCutterAxisX.angle360.inPos AND "Unit1.Em7.ControlNodes".cm.softCam.sepaClampnCutterAxisZ.horizonPos.inPos AND "Unit1.Em7.ControlNodes".cmSepaClampTopUpDown.monitoring.inHomePos AND "Unit1.Em7.ControlNodes".cmSepaClampBottomUpDown.monitoring.inHomePos);
END_REGION

REGION Network 32: Sepa Clamp Job Interface Working Done
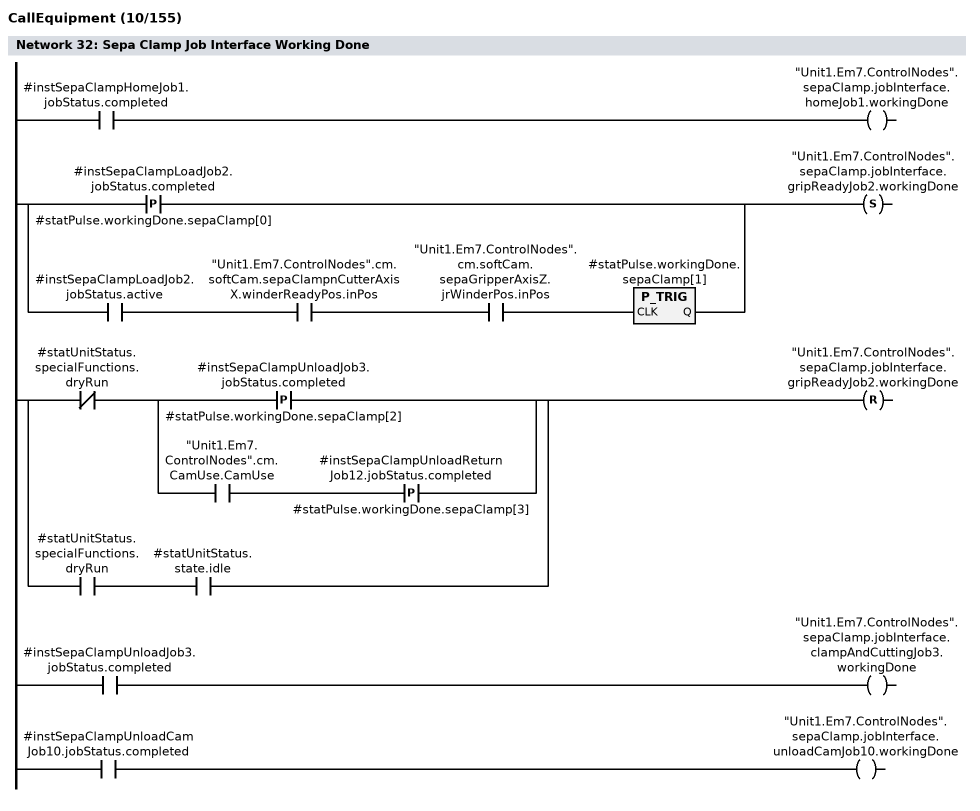
   RUNG wire#powerrail
      Contact( #instSepaClampHomeJob1.jobStatus.completed )
      Coil( "Unit1.Em7.ControlNodes".sepaClamp.jobInterface.homeJob1.workingDone )
   END_RUNG
   RUNG wire#powerrail
      P_Contact(operand := #instSepaClampLoadJob2.jobStatus.completed, bit := #statPulse.workingDone.sepaClamp[0])
      wire#w1
      S_Coil( "Unit1.Em7.ControlNodes".sepaClamp.jobInterface.gripReadyJob2.workingDone )
   END_RUNG
   RUNG wire#powerrail
      Contact( #instSepaClampLoadJob2.jobStatus.active )
      Contact( "Unit1.Em7.ControlNodes".cm.softCam.sepaClampnCutterAxisX.winderReadyPos.inPos )
      Contact( "Unit1.Em7.ControlNodes".cm.softCam.sepaGripperAxisZ.jrWinderPos.inPos )
      P_Trig( #statPulse.workingDone.sepaClamp[1] )
   END_RUNG wire#w1
   RUNG wire#powerrail
      I_Contact( #statUnitStatus.specialFunctions.dryRun )
      wire#w2
      P_Contact(operand := #instSepaClampUnloadJob3.jobStatus.completed, bit := #statPulse.workingDone.sepaClamp[2])
      wire#w3
      R_Coil( "Unit1.Em7.ControlNodes".sepaClamp.jobInterface.gripReadyJob2.workingDone )
   END_RUNG
   RUNG wire#w2
      Contact( "Unit1.Em7.ControlNodes".cm.CamUse.CamUse )
      P_Contact(operand := #instSepaClampUnloadReturnJob12.jobStatus.completed, bit := #statPulse.workingDone.sepaClamp[3])
   END_RUNG wire#w3
   RUNG wire#powerrail
      Contact( #statUnitStatus.specialFunctions.dryRun )
      Contact( #statUnitStatus.state.idle )
   END_RUNG wire#w3
   RUNG wire#powerrail
      Contact( #instSepaClampUnloadJob3.jobStatus.completed )
      Coil( "Unit1.Em7.ControlNodes".sepaClamp.jobInterface.clampAndCuttingJob3.workingDone )
   END_RUNG
   RUNG wire#powerrail
      Contact( #instSepaClampUnloadCamJob10.jobStatus.completed )
      Coil( "Unit1.Em7.ControlNodes".sepaClamp.jobInterface.unloadCamJob10.workingDone )
   END_RUNG
   // the same network as SCL:
   "Unit1.Em7.ControlNodes".sepaClamp.jobInterface.homeJob1.workingDone := #instSepaClampHomeJob1.jobStatus.completed;
   #_w1 := #instSepaClampLoadJob2.jobStatus.completed AND NOT #statPulse.workingDone.sepaClamp[0];   // rising edge of #instSepaClampLoadJob2.jobStatus.completed
   #statPulse.workingDone.sepaClamp[0] := #instSepaClampLoadJob2.jobStatus.completed;
   #_w2 := #instSepaClampLoadJob2.jobStatus.active AND "Unit1.Em7.ControlNodes".cm.softCam.sepaClampnCutterAxisX.winderReadyPos.inPos AND "Unit1.Em7.ControlNodes".cm.softCam.sepaGripperAxisZ.jrWinderPos.inPos;
   #_w3 := #_w2 AND NOT #statPulse.workingDone.sepaClamp[1];   // rising edge
   #statPulse.workingDone.sepaClamp[1] := #_w2;
   IF #_w1 OR #_w3 THEN
       "Unit1.Em7.ControlNodes".sepaClamp.jobInterface.gripReadyJob2.workingDone := TRUE;
   END_IF;
   #_w4 := NOT #statUnitStatus.specialFunctions.dryRun AND #instSepaClampUnloadJob3.jobStatus.completed AND NOT #statPulse.workingDone.sepaClamp[2];   // rising edge of #instSepaClampUnloadJob3.jobStatus.completed
   #statPulse.workingDone.sepaClamp[2] := #instSepaClampUnloadJob3.jobStatus.completed;
   #_w5 := NOT #statUnitStatus.specialFunctions.dryRun AND "Unit1.Em7.ControlNodes".cm.CamUse.CamUse AND #instSepaClampUnloadReturnJob12.jobStatus.completed AND NOT #statPulse.workingDone.sepaClamp[3];   // rising edge of #instSepaClampUnloadReturnJob12.jobStatus.completed
   #statPulse.workingDone.sepaClamp[3] := #instSepaClampUnloadReturnJob12.jobStatus.completed;
   IF #_w4 OR #_w5 OR (#statUnitStatus.specialFunctions.dryRun AND #statUnitStatus.state.idle) THEN
       "Unit1.Em7.ControlNodes".sepaClamp.jobInterface.gripReadyJob2.workingDone := FALSE;
   END_IF;
   "Unit1.Em7.ControlNodes".sepaClamp.jobInterface.clampAndCuttingJob3.workingDone := #instSepaClampUnloadJob3.jobStatus.completed;
   "Unit1.Em7.ControlNodes".sepaClamp.jobInterface.unloadCamJob10.workingDone := #instSepaClampUnloadCamJob10.jobStatus.completed;
END_REGION

REGION Network 33: Sepa Clamp Operation Check
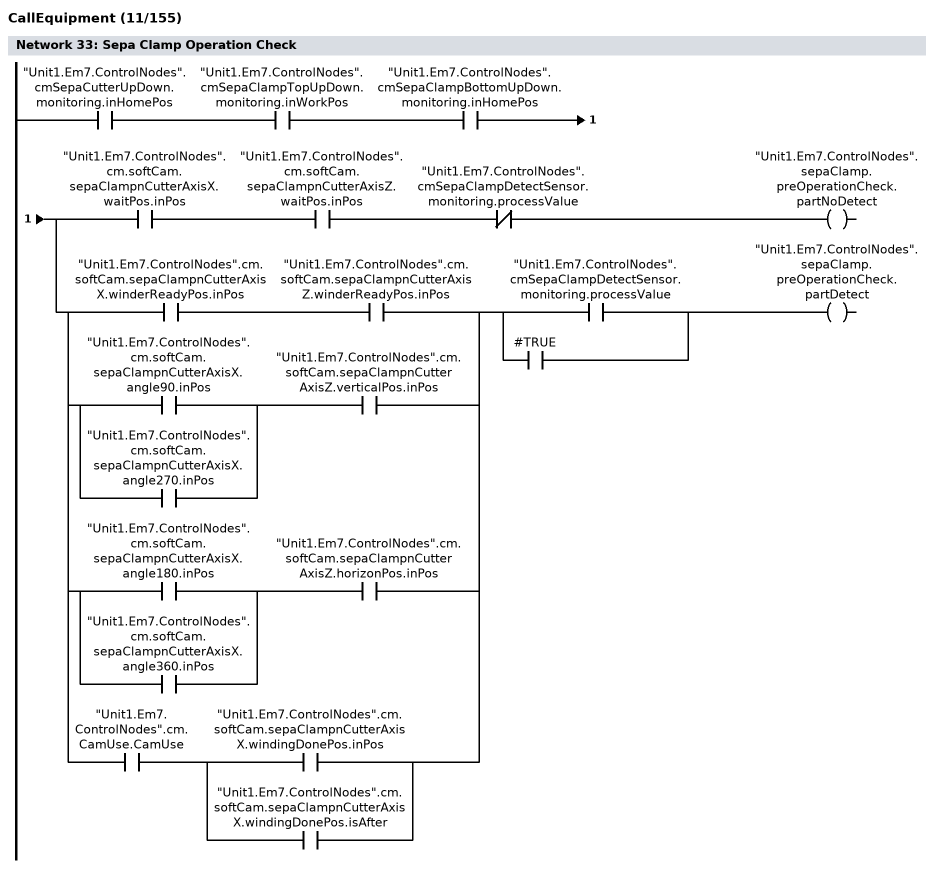
   RUNG wire#powerrail
      Contact( "Unit1.Em7.ControlNodes".cmSepaCutterUpDown.monitoring.inHomePos )
      Contact( "Unit1.Em7.ControlNodes".cmSepaClampTopUpDown.monitoring.inWorkPos )
      Contact( "Unit1.Em7.ControlNodes".cmSepaClampBottomUpDown.monitoring.inHomePos )
      wire#w1
      Contact( "Unit1.Em7.ControlNodes".cm.softCam.sepaClampnCutterAxisX.waitPos.inPos )
      Contact( "Unit1.Em7.ControlNodes".cm.softCam.sepaClampnCutterAxisZ.waitPos.inPos )
      I_Contact( "Unit1.Em7.ControlNodes".cmSepaClampDetectSensor.monitoring.processValue )
      Coil( "Unit1.Em7.ControlNodes".sepaClamp.preOperationCheck.partNoDetect )
   END_RUNG
   RUNG wire#w1
      Contact( "Unit1.Em7.ControlNodes".cm.softCam.sepaClampnCutterAxisX.winderReadyPos.inPos )
      Contact( "Unit1.Em7.ControlNodes".cm.softCam.sepaClampnCutterAxisZ.winderReadyPos.inPos )
      wire#w2
      Contact( "Unit1.Em7.ControlNodes".cmSepaClampDetectSensor.monitoring.processValue )
      wire#w6
      Coil( "Unit1.Em7.ControlNodes".sepaClamp.preOperationCheck.partDetect )
   END_RUNG
   RUNG wire#w1
      Contact( "Unit1.Em7.ControlNodes".cm.softCam.sepaClampnCutterAxisX.angle90.inPos )
      wire#w3
      Contact( "Unit1.Em7.ControlNodes".cm.softCam.sepaClampnCutterAxisZ.verticalPos.inPos )
   END_RUNG wire#w2
   RUNG wire#w1
      Contact( "Unit1.Em7.ControlNodes".cm.softCam.sepaClampnCutterAxisX.angle270.inPos )
   END_RUNG wire#w3
   RUNG wire#w1
      Contact( "Unit1.Em7.ControlNodes".cm.softCam.sepaClampnCutterAxisX.angle180.inPos )
      wire#w4
      Contact( "Unit1.Em7.ControlNodes".cm.softCam.sepaClampnCutterAxisZ.horizonPos.inPos )
   END_RUNG wire#w2
   RUNG wire#w1
      Contact( "Unit1.Em7.ControlNodes".cm.softCam.sepaClampnCutterAxisX.angle360.inPos )
   END_RUNG wire#w4
   RUNG wire#w1
      Contact( "Unit1.Em7.ControlNodes".cm.CamUse.CamUse )
      wire#w5
      Contact( "Unit1.Em7.ControlNodes".cm.softCam.sepaClampnCutterAxisX.windingDonePos.inPos )
   END_RUNG wire#w2
   RUNG wire#w5
      Contact( "Unit1.Em7.ControlNodes".cm.softCam.sepaClampnCutterAxisX.windingDonePos.isAfter )
   END_RUNG wire#w2
   RUNG wire#w2
      Contact( #TRUE )
   END_RUNG wire#w6
   // the same network as SCL:
   #_w1 := "Unit1.Em7.ControlNodes".cmSepaCutterUpDown.monitoring.inHomePos AND "Unit1.Em7.ControlNodes".cmSepaClampTopUpDown.monitoring.inWorkPos AND "Unit1.Em7.ControlNodes".cmSepaClampBottomUpDown.monitoring.inHomePos;
   "Unit1.Em7.ControlNodes".sepaClamp.preOperationCheck.partNoDetect := #_w1 AND "Unit1.Em7.ControlNodes".cm.softCam.sepaClampnCutterAxisX.waitPos.inPos AND "Unit1.Em7.ControlNodes".cm.softCam.sepaClampnCutterAxisZ.waitPos.inPos AND NOT "Unit1.Em7.ControlNodes".cmSepaClampDetectSensor.monitoring.processValue;
   "Unit1.Em7.ControlNodes".sepaClamp.preOperationCheck.partDetect := #_w1 AND (("Unit1.Em7.ControlNodes".cm.softCam.sepaClampnCutterAxisX.winderReadyPos.inPos AND "Unit1.Em7.ControlNodes".cm.softCam.sepaClampnCutterAxisZ.winderReadyPos.inPos) OR (("Unit1.Em7.ControlNodes".cm.softCam.sepaClampnCutterAxisX.angle90.inPos OR "Unit1.Em7.ControlNodes".cm.softCam.sepaClampnCutterAxisX.angle270.inPos) AND "Unit1.Em7.ControlNodes".cm.softCam.sepaClampnCutterAxisZ.verticalPos.inPos) OR (("Unit1.Em7.ControlNodes".cm.softCam.sepaClampnCutterAxisX.angle180.inPos OR "Unit1.Em7.ControlNodes".cm.softCam.sepaClampnCutterAxisX.angle360.inPos) AND "Unit1.Em7.ControlNodes".cm.softCam.sepaClampnCutterAxisZ.horizonPos.inPos) OR ("Unit1.Em7.ControlNodes".cm.CamUse.CamUse AND ("Unit1.Em7.ControlNodes".cm.softCam.sepaClampnCutterAxisX.windingDonePos.inPos OR "Unit1.Em7.ControlNodes".cm.softCam.sepaClampnCutterAxisX.windingDonePos.isAfter))) AND ("Unit1.Em7.ControlNodes".cmSepaClampDetectSensor.monitoring.processValue OR #TRUE);
END_REGION

REGION Network 35: Sepa Gripper Select Job
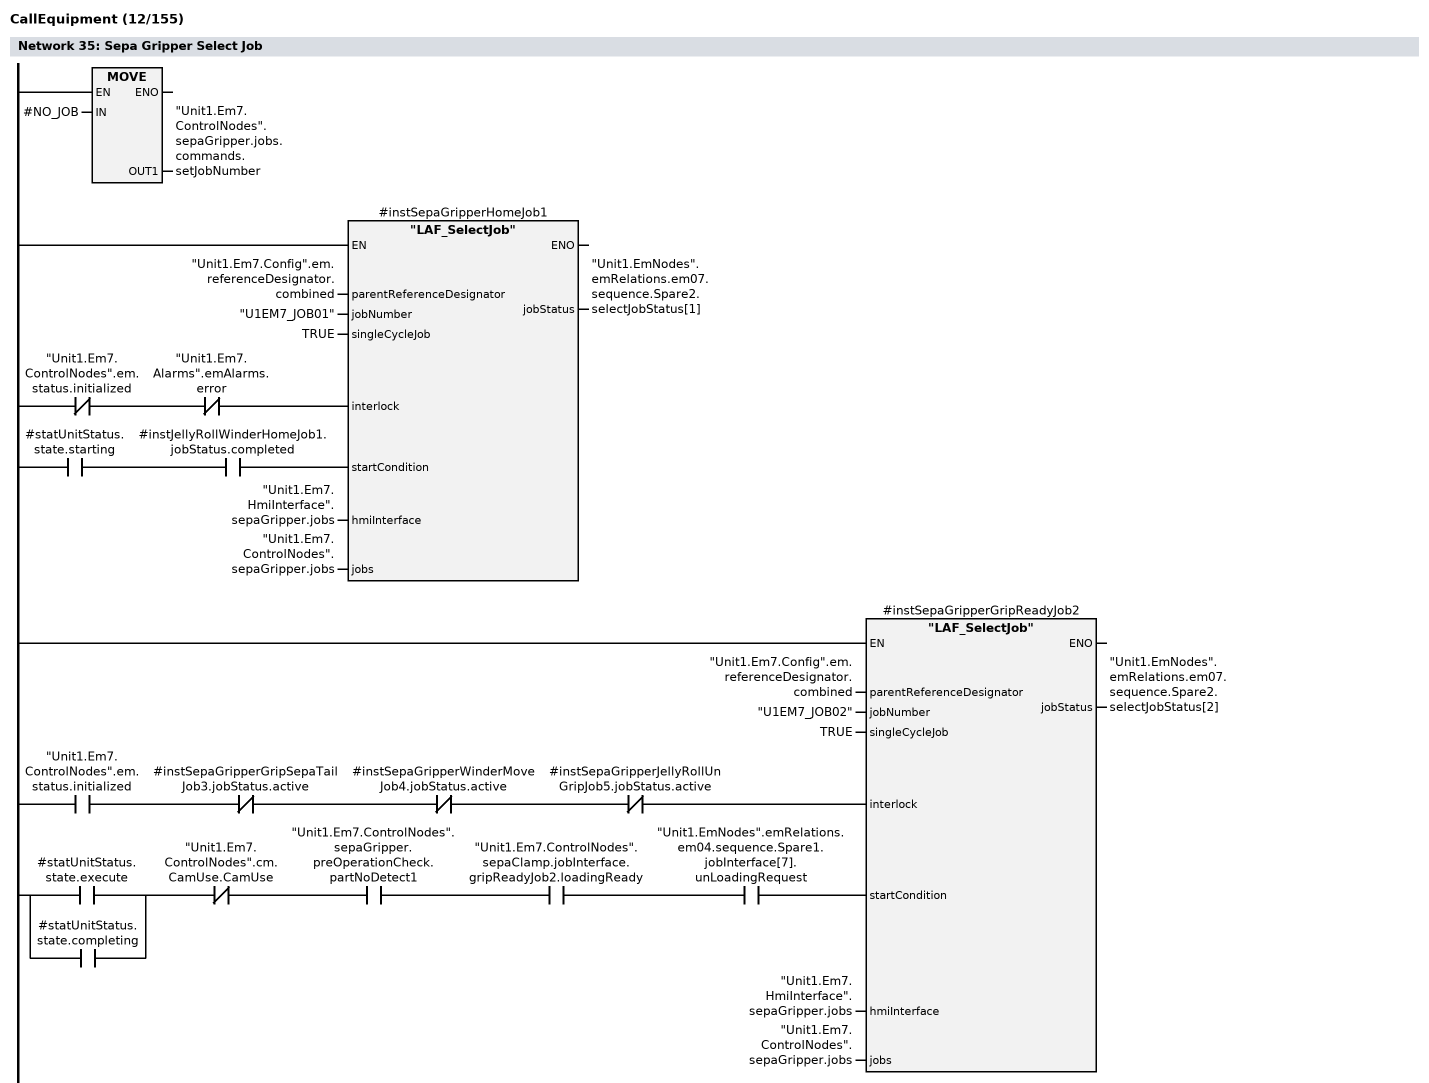
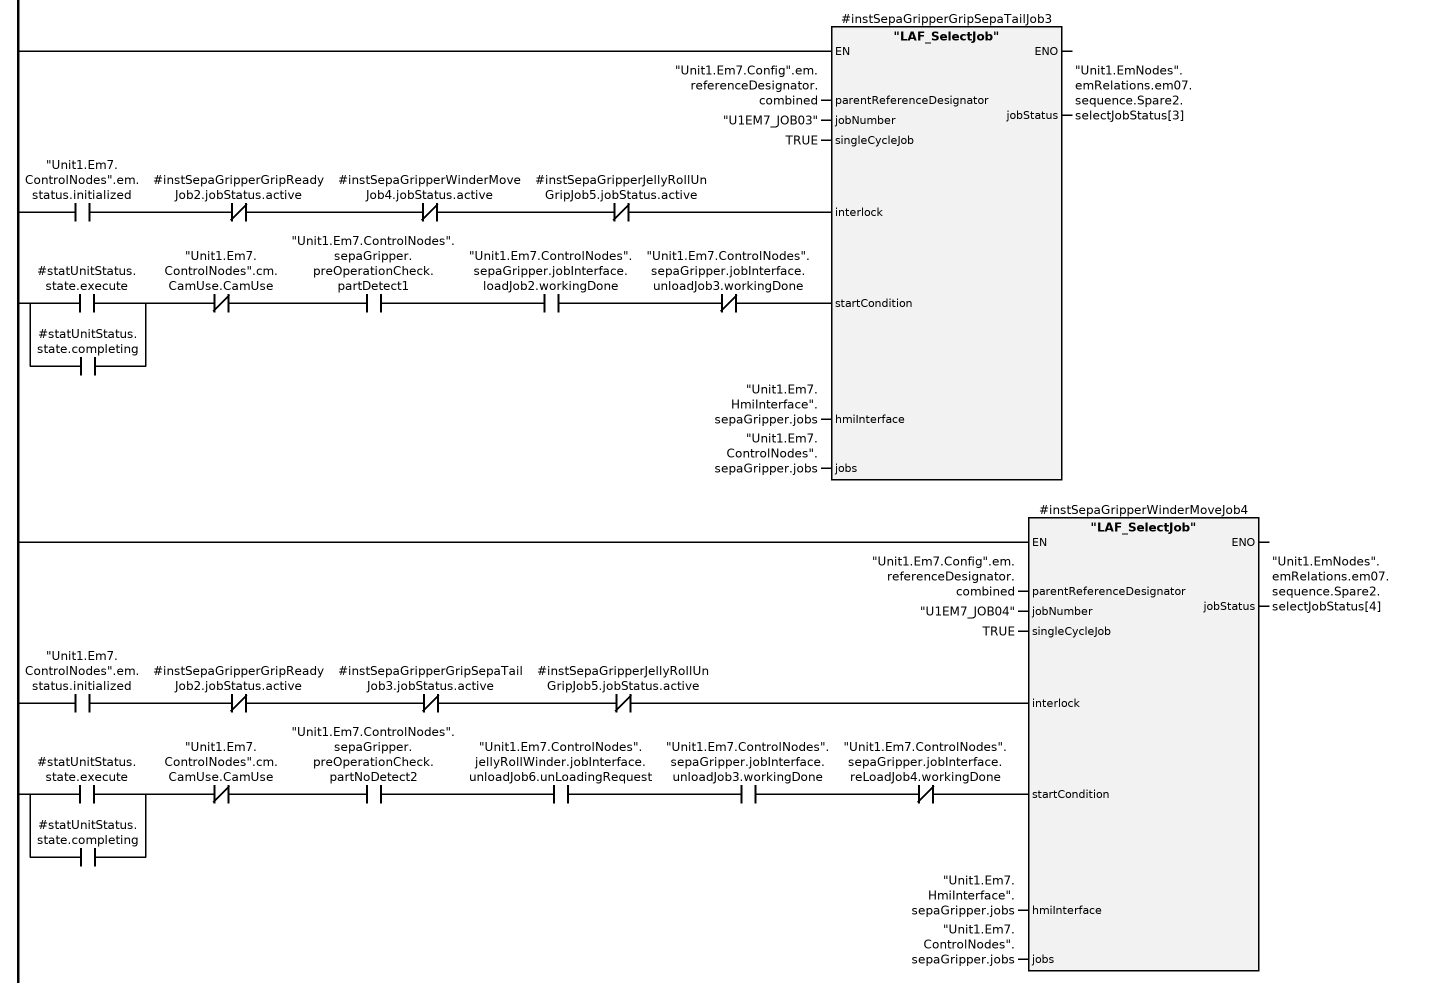
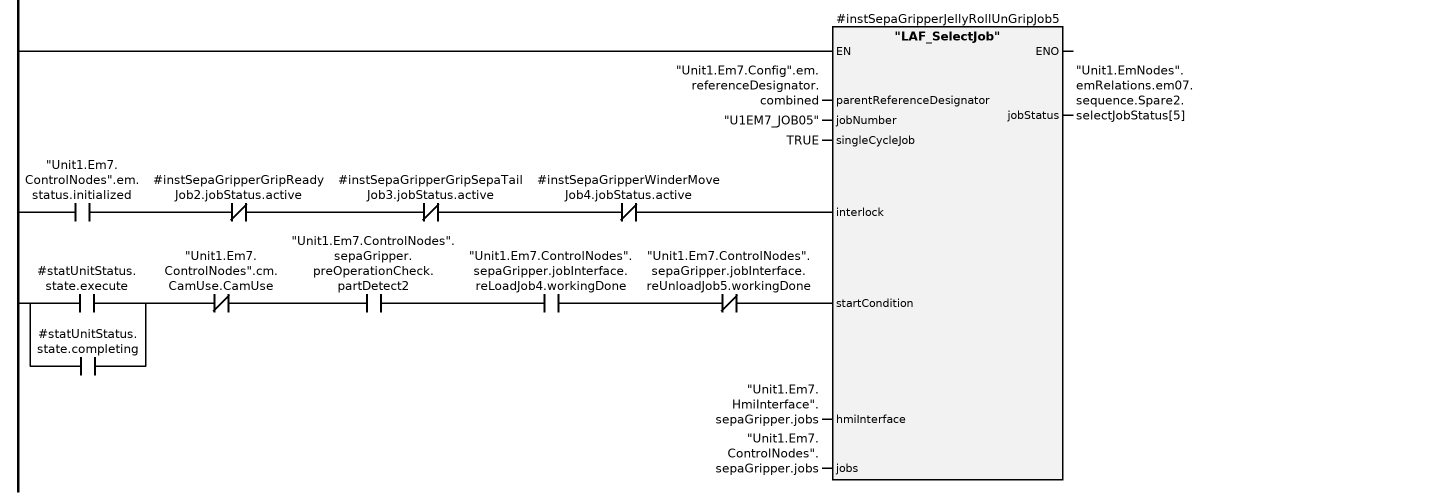
   RUNG wire#powerrail
      Move(in := #NO_JOB, out1 => "Unit1.Em7.ControlNodes".sepaGripper.jobs.commands.setJobNumber)
   END_RUNG
   RUNG wire#powerrail
      #instSepaGripperHomeJob1(interlock := wire#w1, startCondition := wire#w2, parentReferenceDesignator := "Unit1.Em7.Config".em.referenceDesignator.combined, jobNumber := "U1EM7_JOB01", singleCycleJob := TRUE, hmiInterface := "Unit1.Em7.HmiInterface".sepaGripper.jobs, jobs := "Unit1.Em7.ControlNodes".sepaGripper.jobs, jobStatus => "Unit1.EmNodes".emRelations.em07.sequence.Spare2.selectJobStatus[1])
   END_RUNG
   RUNG wire#powerrail
      I_Contact( "Unit1.Em7.ControlNodes".em.status.initialized )
      I_Contact( "Unit1.Em7.Alarms".emAlarms.error )
   END_RUNG wire#w1
   RUNG wire#powerrail
      Contact( #statUnitStatus.state.starting )
      Contact( #instJellyRollWinderHomeJob1.jobStatus.completed )
   END_RUNG wire#w2
   RUNG wire#powerrail
      #instSepaGripperGripReadyJob2(interlock := wire#w3, startCondition := wire#w5, parentReferenceDesignator := "Unit1.Em7.Config".em.referenceDesignator.combined, jobNumber := "U1EM7_JOB02", singleCycleJob := TRUE, hmiInterface := "Unit1.Em7.HmiInterface".sepaGripper.jobs, jobs := "Unit1.Em7.ControlNodes".sepaGripper.jobs, jobStatus => "Unit1.EmNodes".emRelations.em07.sequence.Spare2.selectJobStatus[2])
   END_RUNG
   RUNG wire#powerrail
      Contact( "Unit1.Em7.ControlNodes".em.status.initialized )
      I_Contact( #instSepaGripperGripSepaTailJob3.jobStatus.active )
      I_Contact( #instSepaGripperWinderMoveJob4.jobStatus.active )
      I_Contact( #instSepaGripperJellyRollUnGripJob5.jobStatus.active )
   END_RUNG wire#w3
   RUNG wire#powerrail
      Contact( #statUnitStatus.state.execute )
      wire#w4
      I_Contact( "Unit1.Em7.ControlNodes".cm.CamUse.CamUse )
      Contact( "Unit1.Em7.ControlNodes".sepaGripper.preOperationCheck.partNoDetect1 )
      Contact( "Unit1.Em7.ControlNodes".sepaClamp.jobInterface.gripReadyJob2.loadingReady )
      Contact( "Unit1.EmNodes".emRelations.em04.sequence.Spare1.jobInterface[7].unLoadingRequest )
   END_RUNG wire#w5
   RUNG wire#powerrail
      Contact( #statUnitStatus.state.completing )
   END_RUNG wire#w4
   RUNG wire#powerrail
      #instSepaGripperGripSepaTailJob3(interlock := wire#w6, startCondition := wire#w8, parentReferenceDesignator := "Unit1.Em7.Config".em.referenceDesignator.combined, jobNumber := "U1EM7_JOB03", singleCycleJob := TRUE, hmiInterface := "Unit1.Em7.HmiInterface".sepaGripper.jobs, jobs := "Unit1.Em7.ControlNodes".sepaGripper.jobs, jobStatus => "Unit1.EmNodes".emRelations.em07.sequence.Spare2.selectJobStatus[3])
   END_RUNG
   RUNG wire#powerrail
      Contact( "Unit1.Em7.ControlNodes".em.status.initialized )
      I_Contact( #instSepaGripperGripReadyJob2.jobStatus.active )
      I_Contact( #instSepaGripperWinderMoveJob4.jobStatus.active )
      I_Contact( #instSepaGripperJellyRollUnGripJob5.jobStatus.active )
   END_RUNG wire#w6
   RUNG wire#powerrail
      Contact( #statUnitStatus.state.execute )
      wire#w7
      I_Contact( "Unit1.Em7.ControlNodes".cm.CamUse.CamUse )
      Contact( "Unit1.Em7.ControlNodes".sepaGripper.preOperationCheck.partDetect1 )
      Contact( "Unit1.Em7.ControlNodes".sepaGripper.jobInterface.loadJob2.workingDone )
      I_Contact( "Unit1.Em7.ControlNodes".sepaGripper.jobInterface.unloadJob3.workingDone )
   END_RUNG wire#w8
   RUNG wire#powerrail
      Contact( #statUnitStatus.state.completing )
   END_RUNG wire#w7
   RUNG wire#powerrail
      #instSepaGripperWinderMoveJob4(interlock := wire#w9, startCondition := wire#w11, parentReferenceDesignator := "Unit1.Em7.Config".em.referenceDesignator.combined, jobNumber := "U1EM7_JOB04", singleCycleJob := TRUE, hmiInterface := "Unit1.Em7.HmiInterface".sepaGripper.jobs, jobs := "Unit1.Em7.ControlNodes".sepaGripper.jobs, jobStatus => "Unit1.EmNodes".emRelations.em07.sequence.Spare2.selectJobStatus[4])
   END_RUNG
   RUNG wire#powerrail
      Contact( "Unit1.Em7.ControlNodes".em.status.initialized )
      I_Contact( #instSepaGripperGripReadyJob2.jobStatus.active )
      I_Contact( #instSepaGripperGripSepaTailJob3.jobStatus.active )
      I_Contact( #instSepaGripperJellyRollUnGripJob5.jobStatus.active )
   END_RUNG wire#w9
   RUNG wire#powerrail
      Contact( #statUnitStatus.state.execute )
      wire#w10
      I_Contact( "Unit1.Em7.ControlNodes".cm.CamUse.CamUse )
      Contact( "Unit1.Em7.ControlNodes".sepaGripper.preOperationCheck.partNoDetect2 )
      Contact( "Unit1.Em7.ControlNodes".jellyRollWinder.jobInterface.unloadJob6.unLoadingRequest )
      Contact( "Unit1.Em7.ControlNodes".sepaGripper.jobInterface.unloadJob3.workingDone )
      I_Contact( "Unit1.Em7.ControlNodes".sepaGripper.jobInterface.reLoadJob4.workingDone )
   END_RUNG wire#w11
   RUNG wire#powerrail
      Contact( #statUnitStatus.state.completing )
   END_RUNG wire#w10
   RUNG wire#powerrail
      #instSepaGripperJellyRollUnGripJob5(interlock := wire#w12, startCondition := wire#w14, parentReferenceDesignator := "Unit1.Em7.Config".em.referenceDesignator.combined, jobNumber := "U1EM7_JOB05", singleCycleJob := TRUE, hmiInterface := "Unit1.Em7.HmiInterface".sepaGripper.jobs, jobs := "Unit1.Em7.ControlNodes".sepaGripper.jobs, jobStatus => "Unit1.EmNodes".emRelations.em07.sequence.Spare2.selectJobStatus[5])
   END_RUNG
   RUNG wire#powerrail
      Contact( "Unit1.Em7.ControlNodes".em.status.initialized )
      I_Contact( #instSepaGripperGripReadyJob2.jobStatus.active )
      I_Contact( #instSepaGripperGripSepaTailJob3.jobStatus.active )
      I_Contact( #instSepaGripperWinderMoveJob4.jobStatus.active )
   END_RUNG wire#w12
   RUNG wire#powerrail
      Contact( #statUnitStatus.state.execute )
      wire#w13
      I_Contact( "Unit1.Em7.ControlNodes".cm.CamUse.CamUse )
      Contact( "Unit1.Em7.ControlNodes".sepaGripper.preOperationCheck.partDetect2 )
      Contact( "Unit1.Em7.ControlNodes".sepaGripper.jobInterface.reLoadJob4.workingDone )
      I_Contact( "Unit1.Em7.ControlNodes".sepaGripper.jobInterface.reUnloadJob5.workingDone )
   END_RUNG wire#w14
   RUNG wire#powerrail
      Contact( #statUnitStatus.state.completing )
   END_RUNG wire#w13
   // the same network as SCL:
   "Unit1.Em7.ControlNodes".sepaGripper.jobs.commands.setJobNumber := #NO_JOB;
   #instSepaGripperHomeJob1(parentReferenceDesignator := "Unit1.Em7.Config".em.referenceDesignator.combined,   // "LAF_SelectJob"
                           jobNumber := "U1EM7_JOB01",
                           singleCycleJob := TRUE,
                           interlock := NOT "Unit1.Em7.ControlNodes".em.status.initialized AND NOT "Unit1.Em7.Alarms".emAlarms.error,
                           startCondition := #statUnitStatus.state.starting AND #instJellyRollWinderHomeJob1.jobStatus.completed,
                           hmiInterface := "Unit1.Em7.HmiInterface".sepaGripper.jobs,
                           jobs := "Unit1.Em7.ControlNodes".sepaGripper.jobs,
                           jobStatus => "Unit1.EmNodes".emRelations.em07.sequence.Spare2.selectJobStatus[1]);
   #instSepaGripperGripReadyJob2(parentReferenceDesignator := "Unit1.Em7.Config".em.referenceDesignator.combined,   // "LAF_SelectJob"
                           jobNumber := "U1EM7_JOB02",
                           singleCycleJob := TRUE,
                           interlock := "Unit1.Em7.ControlNodes".em.status.initialized AND NOT #instSepaGripperGripSepaTailJob3.jobStatus.active AND NOT #instSepaGripperWinderMoveJob4.jobStatus.active AND NOT #instSepaGripperJellyRollUnGripJob5.jobStatus.active,
                           startCondition := (#statUnitStatus.state.execute OR #statUnitStatus.state.completing) AND NOT "Unit1.Em7.ControlNodes".cm.CamUse.CamUse AND "Unit1.Em7.ControlNodes".sepaGripper.preOperationCheck.partNoDetect1 AND "Unit1.Em7.ControlNodes".sepaClamp.jobInterface.gripReadyJob2.loadingReady AND "Unit1.EmNodes".emRelations.em04.sequence.Spare1.jobInterface[7].unLoadingRequest,
                           hmiInterface := "Unit1.Em7.HmiInterface".sepaGripper.jobs,
                           jobs := "Unit1.Em7.ControlNodes".sepaGripper.jobs,
                           jobStatus => "Unit1.EmNodes".emRelations.em07.sequence.Spare2.selectJobStatus[2]);
   #instSepaGripperGripSepaTailJob3(parentReferenceDesignator := "Unit1.Em7.Config".em.referenceDesignator.combined,   // "LAF_SelectJob"
                           jobNumber := "U1EM7_JOB03",
                           singleCycleJob := TRUE,
                           interlock := "Unit1.Em7.ControlNodes".em.status.initialized AND NOT #instSepaGripperGripReadyJob2.jobStatus.active AND NOT #instSepaGripperWinderMoveJob4.jobStatus.active AND NOT #instSepaGripperJellyRollUnGripJob5.jobStatus.active,
                           startCondition := (#statUnitStatus.state.execute OR #statUnitStatus.state.completing) AND NOT "Unit1.Em7.ControlNodes".cm.CamUse.CamUse AND "Unit1.Em7.ControlNodes".sepaGripper.preOperationCheck.partDetect1 AND "Unit1.Em7.ControlNodes".sepaGripper.jobInterface.loadJob2.workingDone AND NOT "Unit1.Em7.ControlNodes".sepaGripper.jobInterface.unloadJob3.workingDone,
                           hmiInterface := "Unit1.Em7.HmiInterface".sepaGripper.jobs,
                           jobs := "Unit1.Em7.ControlNodes".sepaGripper.jobs,
                           jobStatus => "Unit1.EmNodes".emRelations.em07.sequence.Spare2.selectJobStatus[3]);
   #instSepaGripperWinderMoveJob4(parentReferenceDesignator := "Unit1.Em7.Config".em.referenceDesignator.combined,   // "LAF_SelectJob"
                           jobNumber := "U1EM7_JOB04",
                           singleCycleJob := TRUE,
                           interlock := "Unit1.Em7.ControlNodes".em.status.initialized AND NOT #instSepaGripperGripReadyJob2.jobStatus.active AND NOT #instSepaGripperGripSepaTailJob3.jobStatus.active AND NOT #instSepaGripperJellyRollUnGripJob5.jobStatus.active,
                           startCondition := (#statUnitStatus.state.execute OR #statUnitStatus.state.completing) AND NOT "Unit1.Em7.ControlNodes".cm.CamUse.CamUse AND "Unit1.Em7.ControlNodes".sepaGripper.preOperationCheck.partNoDetect2 AND "Unit1.Em7.ControlNodes".jellyRollWinder.jobInterface.unloadJob6.unLoadingRequest AND "Unit1.Em7.ControlNodes".sepaGripper.jobInterface.unloadJob3.workingDone AND NOT "Unit1.Em7.ControlNodes".sepaGripper.jobInterface.reLoadJob4.workingDone,
                           hmiInterface := "Unit1.Em7.HmiInterface".sepaGripper.jobs,
                           jobs := "Unit1.Em7.ControlNodes".sepaGripper.jobs,
                           jobStatus => "Unit1.EmNodes".emRelations.em07.sequence.Spare2.selectJobStatus[4]);
   #instSepaGripperJellyRollUnGripJob5(parentReferenceDesignator := "Unit1.Em7.Config".em.referenceDesignator.combined,   // "LAF_SelectJob"
                           jobNumber := "U1EM7_JOB05",
                           singleCycleJob := TRUE,
                           interlock := "Unit1.Em7.ControlNodes".em.status.initialized AND NOT #instSepaGripperGripReadyJob2.jobStatus.active AND NOT #instSepaGripperGripSepaTailJob3.jobStatus.active AND NOT #instSepaGripperWinderMoveJob4.jobStatus.active,
                           startCondition := (#statUnitStatus.state.execute OR #statUnitStatus.state.completing) AND NOT "Unit1.Em7.ControlNodes".cm.CamUse.CamUse AND "Unit1.Em7.ControlNodes".sepaGripper.preOperationCheck.partDetect2 AND "Unit1.Em7.ControlNodes".sepaGripper.jobInterface.reLoadJob4.workingDone AND NOT "Unit1.Em7.ControlNodes".sepaGripper.jobInterface.reUnloadJob5.workingDone,
                           hmiInterface := "Unit1.Em7.HmiInterface".sepaGripper.jobs,
                           jobs := "Unit1.Em7.ControlNodes".sepaGripper.jobs,
                           jobStatus => "Unit1.EmNodes".emRelations.em07.sequence.Spare2.selectJobStatus[5]);
END_REGION

REGION Network 36: Sepa Gripper Select Job [Cam]
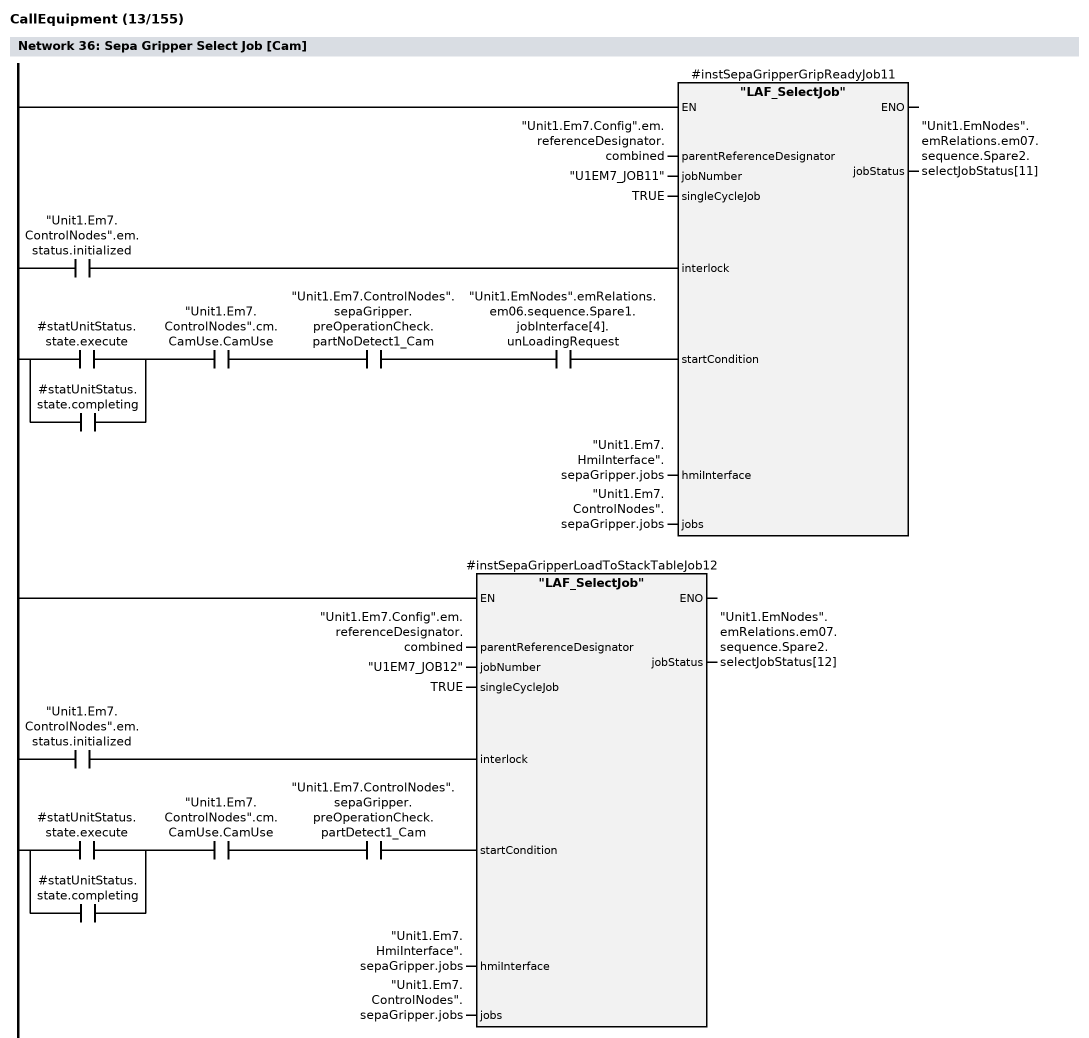
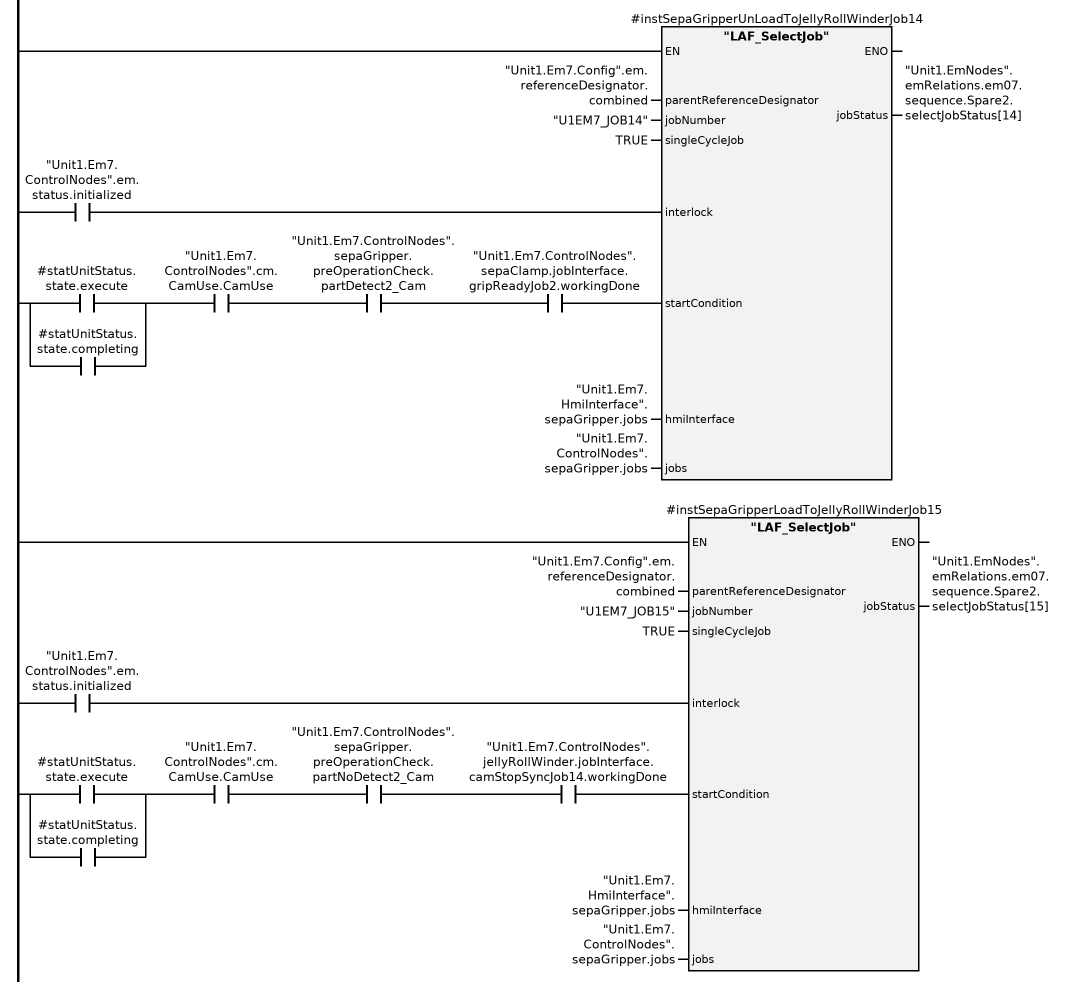
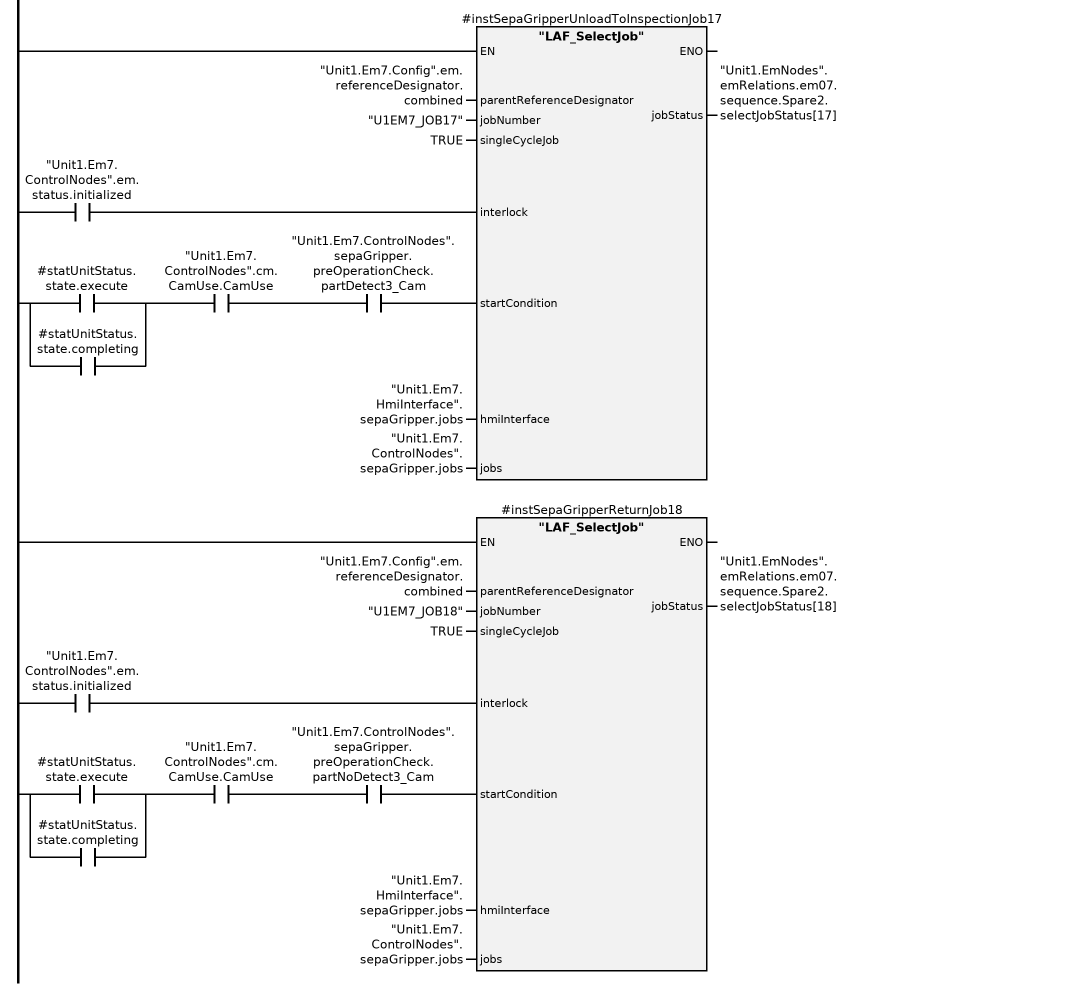
   RUNG wire#powerrail
      #instSepaGripperGripReadyJob11(interlock := wire#w1, startCondition := wire#w3, parentReferenceDesignator := "Unit1.Em7.Config".em.referenceDesignator.combined, jobNumber := "U1EM7_JOB11", singleCycleJob := TRUE, hmiInterface := "Unit1.Em7.HmiInterface".sepaGripper.jobs, jobs := "Unit1.Em7.ControlNodes".sepaGripper.jobs, jobStatus => "Unit1.EmNodes".emRelations.em07.sequence.Spare2.selectJobStatus[11])
   END_RUNG
   RUNG wire#powerrail
      Contact( "Unit1.Em7.ControlNodes".em.status.initialized )
   END_RUNG wire#w1
   RUNG wire#powerrail
      Contact( #statUnitStatus.state.execute )
      wire#w2
      Contact( "Unit1.Em7.ControlNodes".cm.CamUse.CamUse )
      Contact( "Unit1.Em7.ControlNodes".sepaGripper.preOperationCheck.partNoDetect1_Cam )
      Contact( "Unit1.EmNodes".emRelations.em06.sequence.Spare1.jobInterface[4].unLoadingRequest )
   END_RUNG wire#w3
   RUNG wire#powerrail
      Contact( #statUnitStatus.state.completing )
   END_RUNG wire#w2
   RUNG wire#powerrail
      #instSepaGripperLoadToStackTableJob12(interlock := wire#w4, startCondition := wire#w6, parentReferenceDesignator := "Unit1.Em7.Config".em.referenceDesignator.combined, jobNumber := "U1EM7_JOB12", singleCycleJob := TRUE, hmiInterface := "Unit1.Em7.HmiInterface".sepaGripper.jobs, jobs := "Unit1.Em7.ControlNodes".sepaGripper.jobs, jobStatus => "Unit1.EmNodes".emRelations.em07.sequence.Spare2.selectJobStatus[12])
   END_RUNG
   RUNG wire#powerrail
      Contact( "Unit1.Em7.ControlNodes".em.status.initialized )
   END_RUNG wire#w4
   RUNG wire#powerrail
      Contact( #statUnitStatus.state.execute )
      wire#w5
      Contact( "Unit1.Em7.ControlNodes".cm.CamUse.CamUse )
      Contact( "Unit1.Em7.ControlNodes".sepaGripper.preOperationCheck.partDetect1_Cam )
   END_RUNG wire#w6
   RUNG wire#powerrail
      Contact( #statUnitStatus.state.completing )
   END_RUNG wire#w5
   RUNG wire#powerrail
      #instSepaGripperUnLoadToJellyRollWinderJob14(interlock := wire#w7, startCondition := wire#w9, parentReferenceDesignator := "Unit1.Em7.Config".em.referenceDesignator.combined, jobNumber := "U1EM7_JOB14", singleCycleJob := TRUE, hmiInterface := "Unit1.Em7.HmiInterface".sepaGripper.jobs, jobs := "Unit1.Em7.ControlNodes".sepaGripper.jobs, jobStatus => "Unit1.EmNodes".emRelations.em07.sequence.Spare2.selectJobStatus[14])
   END_RUNG
   RUNG wire#powerrail
      Contact( "Unit1.Em7.ControlNodes".em.status.initialized )
   END_RUNG wire#w7
   RUNG wire#powerrail
      Contact( #statUnitStatus.state.execute )
      wire#w8
      Contact( "Unit1.Em7.ControlNodes".cm.CamUse.CamUse )
      Contact( "Unit1.Em7.ControlNodes".sepaGripper.preOperationCheck.partDetect2_Cam )
      Contact( "Unit1.Em7.ControlNodes".sepaClamp.jobInterface.gripReadyJob2.workingDone )
   END_RUNG wire#w9
   RUNG wire#powerrail
      Contact( #statUnitStatus.state.completing )
   END_RUNG wire#w8
   RUNG wire#powerrail
      #instSepaGripperLoadToJellyRollWinderJob15(interlock := wire#w10, startCondition := wire#w12, parentReferenceDesignator := "Unit1.Em7.Config".em.referenceDesignator.combined, jobNumber := "U1EM7_JOB15", singleCycleJob := TRUE, hmiInterface := "Unit1.Em7.HmiInterface".sepaGripper.jobs, jobs := "Unit1.Em7.ControlNodes".sepaGripper.jobs, jobStatus => "Unit1.EmNodes".emRelations.em07.sequence.Spare2.selectJobStatus[15])
   END_RUNG
   RUNG wire#powerrail
      Contact( "Unit1.Em7.ControlNodes".em.status.initialized )
   END_RUNG wire#w10
   RUNG wire#powerrail
      Contact( #statUnitStatus.state.execute )
      wire#w11
      Contact( "Unit1.Em7.ControlNodes".cm.CamUse.CamUse )
      Contact( "Unit1.Em7.ControlNodes".sepaGripper.preOperationCheck.partNoDetect2_Cam )
      Contact( "Unit1.Em7.ControlNodes".jellyRollWinder.jobInterface.camStopSyncJob14.workingDone )
   END_RUNG wire#w12
   RUNG wire#powerrail
      Contact( #statUnitStatus.state.completing )
   END_RUNG wire#w11
   RUNG wire#powerrail
      #instSepaGripperUnloadToInspectionJob17(interlock := wire#w13, startCondition := wire#w15, parentReferenceDesignator := "Unit1.Em7.Config".em.referenceDesignator.combined, jobNumber := "U1EM7_JOB17", singleCycleJob := TRUE, hmiInterface := "Unit1.Em7.HmiInterface".sepaGripper.jobs, jobs := "Unit1.Em7.ControlNodes".sepaGripper.jobs, jobStatus => "Unit1.EmNodes".emRelations.em07.sequence.Spare2.selectJobStatus[17])
   END_RUNG
   RUNG wire#powerrail
      Contact( "Unit1.Em7.ControlNodes".em.status.initialized )
   END_RUNG wire#w13
   RUNG wire#powerrail
      Contact( #statUnitStatus.state.execute )
      wire#w14
      Contact( "Unit1.Em7.ControlNodes".cm.CamUse.CamUse )
      Contact( "Unit1.Em7.ControlNodes".sepaGripper.preOperationCheck.partDetect3_Cam )
   END_RUNG wire#w15
   RUNG wire#powerrail
      Contact( #statUnitStatus.state.completing )
   END_RUNG wire#w14
   RUNG wire#powerrail
      #instSepaGripperReturnJob18(interlock := wire#w16, startCondition := wire#w18, parentReferenceDesignator := "Unit1.Em7.Config".em.referenceDesignator.combined, jobNumber := "U1EM7_JOB18", singleCycleJob := TRUE, hmiInterface := "Unit1.Em7.HmiInterface".sepaGripper.jobs, jobs := "Unit1.Em7.ControlNodes".sepaGripper.jobs, jobStatus => "Unit1.EmNodes".emRelations.em07.sequence.Spare2.selectJobStatus[18])
   END_RUNG
   RUNG wire#powerrail
      Contact( "Unit1.Em7.ControlNodes".em.status.initialized )
   END_RUNG wire#w16
   RUNG wire#powerrail
      Contact( #statUnitStatus.state.execute )
      wire#w17
      Contact( "Unit1.Em7.ControlNodes".cm.CamUse.CamUse )
      Contact( "Unit1.Em7.ControlNodes".sepaGripper.preOperationCheck.partNoDetect3_Cam )
   END_RUNG wire#w18
   RUNG wire#powerrail
      Contact( #statUnitStatus.state.completing )
   END_RUNG wire#w17
   // the same network as SCL:
   #instSepaGripperGripReadyJob11(parentReferenceDesignator := "Unit1.Em7.Config".em.referenceDesignator.combined,   // "LAF_SelectJob"
                           jobNumber := "U1EM7_JOB11",
                           singleCycleJob := TRUE,
                           interlock := "Unit1.Em7.ControlNodes".em.status.initialized,
                           startCondition := (#statUnitStatus.state.execute OR #statUnitStatus.state.completing) AND "Unit1.Em7.ControlNodes".cm.CamUse.CamUse AND "Unit1.Em7.ControlNodes".sepaGripper.preOperationCheck.partNoDetect1_Cam AND "Unit1.EmNodes".emRelations.em06.sequence.Spare1.jobInterface[4].unLoadingRequest,
                           hmiInterface := "Unit1.Em7.HmiInterface".sepaGripper.jobs,
                           jobs := "Unit1.Em7.ControlNodes".sepaGripper.jobs,
                           jobStatus => "Unit1.EmNodes".emRelations.em07.sequence.Spare2.selectJobStatus[11]);
   #instSepaGripperLoadToStackTableJob12(parentReferenceDesignator := "Unit1.Em7.Config".em.referenceDesignator.combined,   // "LAF_SelectJob"
                           jobNumber := "U1EM7_JOB12",
                           singleCycleJob := TRUE,
                           interlock := "Unit1.Em7.ControlNodes".em.status.initialized,
                           startCondition := (#statUnitStatus.state.execute OR #statUnitStatus.state.completing) AND "Unit1.Em7.ControlNodes".cm.CamUse.CamUse AND "Unit1.Em7.ControlNodes".sepaGripper.preOperationCheck.partDetect1_Cam,
                           hmiInterface := "Unit1.Em7.HmiInterface".sepaGripper.jobs,
                           jobs := "Unit1.Em7.ControlNodes".sepaGripper.jobs,
                           jobStatus => "Unit1.EmNodes".emRelations.em07.sequence.Spare2.selectJobStatus[12]);
   #instSepaGripperUnLoadToJellyRollWinderJob14(parentReferenceDesignator := "Unit1.Em7.Config".em.referenceDesignator.combined,   // "LAF_SelectJob"
                           jobNumber := "U1EM7_JOB14",
                           singleCycleJob := TRUE,
                           interlock := "Unit1.Em7.ControlNodes".em.status.initialized,
                           startCondition := (#statUnitStatus.state.execute OR #statUnitStatus.state.completing) AND "Unit1.Em7.ControlNodes".cm.CamUse.CamUse AND "Unit1.Em7.ControlNodes".sepaGripper.preOperationCheck.partDetect2_Cam AND "Unit1.Em7.ControlNodes".sepaClamp.jobInterface.gripReadyJob2.workingDone,
                           hmiInterface := "Unit1.Em7.HmiInterface".sepaGripper.jobs,
                           jobs := "Unit1.Em7.ControlNodes".sepaGripper.jobs,
                           jobStatus => "Unit1.EmNodes".emRelations.em07.sequence.Spare2.selectJobStatus[14]);
   #instSepaGripperLoadToJellyRollWinderJob15(parentReferenceDesignator := "Unit1.Em7.Config".em.referenceDesignator.combined,   // "LAF_SelectJob"
                           jobNumber := "U1EM7_JOB15",
                           singleCycleJob := TRUE,
                           interlock := "Unit1.Em7.ControlNodes".em.status.initialized,
                           startCondition := (#statUnitStatus.state.execute OR #statUnitStatus.state.completing) AND "Unit1.Em7.ControlNodes".cm.CamUse.CamUse AND "Unit1.Em7.ControlNodes".sepaGripper.preOperationCheck.partNoDetect2_Cam AND "Unit1.Em7.ControlNodes".jellyRollWinder.jobInterface.camStopSyncJob14.workingDone,
                           hmiInterface := "Unit1.Em7.HmiInterface".sepaGripper.jobs,
                           jobs := "Unit1.Em7.ControlNodes".sepaGripper.jobs,
                           jobStatus => "Unit1.EmNodes".emRelations.em07.sequence.Spare2.selectJobStatus[15]);
   #instSepaGripperUnloadToInspectionJob17(parentReferenceDesignator := "Unit1.Em7.Config".em.referenceDesignator.combined,   // "LAF_SelectJob"
                           jobNumber := "U1EM7_JOB17",
                           singleCycleJob := TRUE,
                           interlock := "Unit1.Em7.ControlNodes".em.status.initialized,
                           startCondition := (#statUnitStatus.state.execute OR #statUnitStatus.state.completing) AND "Unit1.Em7.ControlNodes".cm.CamUse.CamUse AND "Unit1.Em7.ControlNodes".sepaGripper.preOperationCheck.partDetect3_Cam,
                           hmiInterface := "Unit1.Em7.HmiInterface".sepaGripper.jobs,
                           jobs := "Unit1.Em7.ControlNodes".sepaGripper.jobs,
                           jobStatus => "Unit1.EmNodes".emRelations.em07.sequence.Spare2.selectJobStatus[17]);
   #instSepaGripperReturnJob18(parentReferenceDesignator := "Unit1.Em7.Config".em.referenceDesignator.combined,   // "LAF_SelectJob"
                           jobNumber := "U1EM7_JOB18",
                           singleCycleJob := TRUE,
                           interlock := "Unit1.Em7.ControlNodes".em.status.initialized,
                           startCondition := (#statUnitStatus.state.execute OR #statUnitStatus.state.completing) AND "Unit1.Em7.ControlNodes".cm.CamUse.CamUse AND "Unit1.Em7.ControlNodes".sepaGripper.preOperationCheck.partNoDetect3_Cam,
                           hmiInterface := "Unit1.Em7.HmiInterface".sepaGripper.jobs,
                           jobs := "Unit1.Em7.ControlNodes".sepaGripper.jobs,
                           jobStatus => "Unit1.EmNodes".emRelations.em07.sequence.Spare2.selectJobStatus[18]);
END_REGION

REGION Network 37: Sepa Gripper Job Interface [Loading]
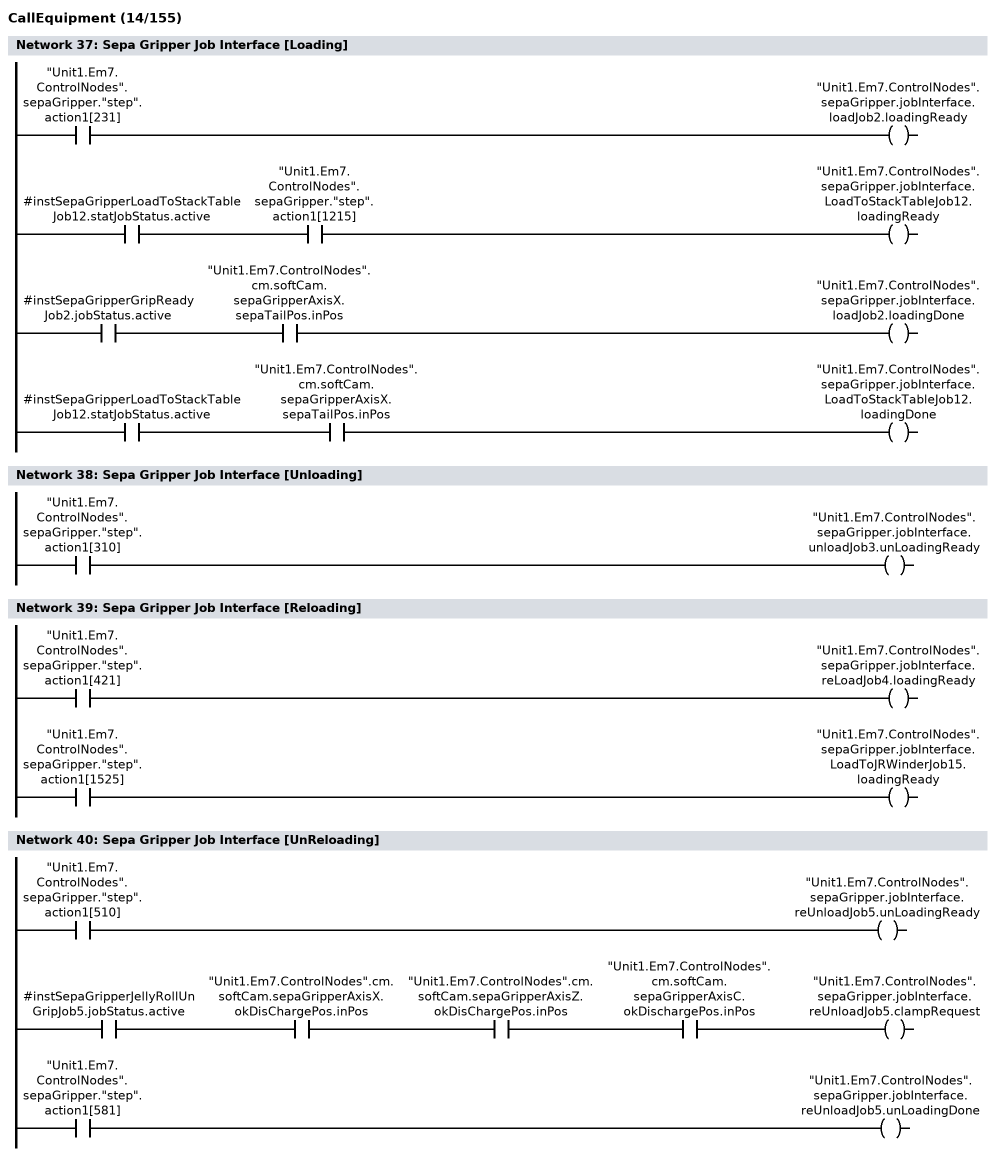
   RUNG wire#powerrail
      Contact( "Unit1.Em7.ControlNodes".sepaGripper."step".action1[231] )
      Coil( "Unit1.Em7.ControlNodes".sepaGripper.jobInterface.loadJob2.loadingReady )
   END_RUNG
   RUNG wire#powerrail
      Contact( #instSepaGripperLoadToStackTableJob12.statJobStatus.active )
      Contact( "Unit1.Em7.ControlNodes".sepaGripper."step".action1[1215] )
      Coil( "Unit1.Em7.ControlNodes".sepaGripper.jobInterface.LoadToStackTableJob12.loadingReady )
   END_RUNG
   RUNG wire#powerrail
      Contact( #instSepaGripperGripReadyJob2.jobStatus.active )
      Contact( "Unit1.Em7.ControlNodes".cm.softCam.sepaGripperAxisX.sepaTailPos.inPos )
      Coil( "Unit1.Em7.ControlNodes".sepaGripper.jobInterface.loadJob2.loadingDone )
   END_RUNG
   RUNG wire#powerrail
      Contact( #instSepaGripperLoadToStackTableJob12.statJobStatus.active )
      Contact( "Unit1.Em7.ControlNodes".cm.softCam.sepaGripperAxisX.sepaTailPos.inPos )
      Coil( "Unit1.Em7.ControlNodes".sepaGripper.jobInterface.LoadToStackTableJob12.loadingDone )
   END_RUNG
   // the same network as SCL:
   "Unit1.Em7.ControlNodes".sepaGripper.jobInterface.loadJob2.loadingReady := "Unit1.Em7.ControlNodes".sepaGripper."step".action1[231];
   "Unit1.Em7.ControlNodes".sepaGripper.jobInterface.LoadToStackTableJob12.loadingReady := #instSepaGripperLoadToStackTableJob12.statJobStatus.active AND "Unit1.Em7.ControlNodes".sepaGripper."step".action1[1215];
   "Unit1.Em7.ControlNodes".sepaGripper.jobInterface.loadJob2.loadingDone := #instSepaGripperGripReadyJob2.jobStatus.active AND "Unit1.Em7.ControlNodes".cm.softCam.sepaGripperAxisX.sepaTailPos.inPos;
   "Unit1.Em7.ControlNodes".sepaGripper.jobInterface.LoadToStackTableJob12.loadingDone := #instSepaGripperLoadToStackTableJob12.statJobStatus.active AND "Unit1.Em7.ControlNodes".cm.softCam.sepaGripperAxisX.sepaTailPos.inPos;
END_REGION

REGION Network 38: Sepa Gripper Job Interface [Unloading]
   RUNG wire#powerrail
      Contact( "Unit1.Em7.ControlNodes".sepaGripper."step".action1[310] )
      Coil( "Unit1.Em7.ControlNodes".sepaGripper.jobInterface.unloadJob3.unLoadingReady )
   END_RUNG
   // the same network as SCL:
   "Unit1.Em7.ControlNodes".sepaGripper.jobInterface.unloadJob3.unLoadingReady := "Unit1.Em7.ControlNodes".sepaGripper."step".action1[310];
END_REGION

REGION Network 39: Sepa Gripper Job Interface [Reloading]
   RUNG wire#powerrail
      Contact( "Unit1.Em7.ControlNodes".sepaGripper."step".action1[421] )
      Coil( "Unit1.Em7.ControlNodes".sepaGripper.jobInterface.reLoadJob4.loadingReady )
   END_RUNG
   RUNG wire#powerrail
      Contact( "Unit1.Em7.ControlNodes".sepaGripper."step".action1[1525] )
      Coil( "Unit1.Em7.ControlNodes".sepaGripper.jobInterface.LoadToJRWinderJob15.loadingReady )
   END_RUNG
   // the same network as SCL:
   "Unit1.Em7.ControlNodes".sepaGripper.jobInterface.reLoadJob4.loadingReady := "Unit1.Em7.ControlNodes".sepaGripper."step".action1[421];
   "Unit1.Em7.ControlNodes".sepaGripper.jobInterface.LoadToJRWinderJob15.loadingReady := "Unit1.Em7.ControlNodes".sepaGripper."step".action1[1525];
END_REGION

